    !Tr_meulage_bavure : Meulage de la bavure
    LOCAL CONST Robtarget Tr_meulage_bavure_0 := [[-118.3383671875,-114.213265625,120.94103125],[0.686050855165754,-0.669480714392343,0.19893041187492,-0.203854086086913],[0,0,0,0],[8.999999E+09,8.999999E+09,8.999999E+09,8.999999E+09,8.999999E+09,8.999999E+09]];
    LOCAL CONST Robtarget Tr_meulage_bavure_1 := [[-119.6316875,-113.9973125,120.9542265625],[0.684325266912173,-0.667622761472622,0.204761653370109,-0.209884355630412],[0,0,0,0],[8.999999E+09,8.999999E+09,8.999999E+09,8.999999E+09,8.999999E+09,8.999999E+09]];
    LOCAL CONST Robtarget Tr_meulage_bavure_2 := [[-123.489203125,-113.0502109375,120.9455703125],[0.678831233917672,-0.66176958949123,0.222117553220813,-0.227844154705838],[0,0,0,0],[8.999999E+09,8.999999E+09,8.999999E+09,8.999999E+09,8.999999E+09,8.999999E+09]];
    LOCAL CONST Robtarget Tr_meulage_bavure_3 := [[-123.584859375,-113.0222734375,120.9446484375],[0.668624934223721,-0.651045700458164,0.250641046300353,-0.257408739476203],[0,0,0,0],[8.999999E+09,8.999999E+09,8.999999E+09,8.999999E+09,8.999999E+09,8.999999E+09]];
    LOCAL CONST Robtarget Tr_meulage_bavure_4 := [[-125.8031953125,-111.60703125,120.8016875],[0.652172819034723,-0.634001173456056,0.28968410592264,-0.297986987877738],[0,0,0,0],[8.999999E+09,8.999999E+09,8.999999E+09,8.999999E+09,8.999999E+09,8.999999E+09]];
    LOCAL CONST Robtarget Tr_meulage_bavure_5 := [[-126.4752265625,-111.0076484375,120.7313359375],[0.627744539207993,-0.609028304977179,0.337572017036929,-0.347946045450712],[0,0,0,0],[8.999999E+09,8.999999E+09,8.999999E+09,8.999999E+09,8.999999E+09,8.999999E+09]];
    LOCAL CONST Robtarget Tr_meulage_bavure_6 := [[-126.8417890625,-109.187203125,120.45625],[0.594928081420455,-0.575888879676794,0.389993371636008,-0.402886766079456],[0,0,0,0],[8.999999E+09,8.999999E+09,8.999999E+09,8.999999E+09,8.999999E+09,8.999999E+09]];
    LOCAL CONST Robtarget Tr_meulage_bavure_7 := [[-127.4551015625,-107.313234375,120.181734375],[0.55678322484501,-0.537637245657738,0.439837894187461,-0.455501108066151],[0,0,0,0],[8.999999E+09,8.999999E+09,8.999999E+09,8.999999E+09,8.999999E+09,8.999999E+09]];
    LOCAL CONST Robtarget Tr_meulage_bavure_8 := [[-126.9923671875,-103.8465,119.6153203125],[0.519549603690322,-0.500370572095961,0.48044926250951,-0.498864717172559],[0,0,0,0],[8.999999E+09,8.999999E+09,8.999999E+09,8.999999E+09,8.999999E+09,8.999999E+09]];
    LOCAL CONST Robtarget Tr_meulage_bavure_9 := [[-126.982359375,-103.7414453125,119.5983046875],[0.489009720279578,-0.469707644324052,0.509165648687706,-0.530089204315714],[0,0,0,0],[8.999999E+09,8.999999E+09,8.999999E+09,8.999999E+09,8.999999E+09,8.999999E+09]];
    LOCAL CONST Robtarget Tr_meulage_bavure_10 := [[-126.968546875,-103.6983828125,119.5909765625],[0.467640365028404,-0.44800873567007,0.527122282578491,-0.550220647530287],[0,0,0,0],[8.999999E+09,8.999999E+09,8.999999E+09,8.999999E+09,8.999999E+09,8.999999E+09]];
    LOCAL CONST Robtarget Tr_meulage_bavure_11 := [[-126.9365390625,-103.55375,119.566875],[0.454927941273034,-0.434723512970439,0.536951278731924,-0.561906896013807],[0,0,0,0],[8.999999E+09,8.999999E+09,8.999999E+09,8.999999E+09,8.999999E+09,8.999999E+09]];
    LOCAL CONST Robtarget Tr_meulage_bavure_12 := [[-125.41084375,-97.252625,118.5122578125],[0.448816582731819,-0.427864419149345,0.541337479198651,-0.567846323846318],[0,0,0,0],[8.999999E+09,8.999999E+09,8.999999E+09,8.999999E+09,8.999999E+09,8.999999E+09]];
    LOCAL CONST Robtarget Tr_meulage_bavure_13 := [[-124.5225390625,-93.8810859375,117.945328125],[0.446998595891194,-0.425203405993345,0.54242876260288,-0.570232721179755],[0,0,0,0],[8.999999E+09,8.999999E+09,8.999999E+09,8.999999E+09,8.999999E+09,8.999999E+09]];
    LOCAL CONST Robtarget Tr_meulage_bavure_14 := [[-123.5930703125,-90.2569375,117.3368515625],[0.447502976011157,-0.424854620024497,0.541806054841724,-0.570688914595198],[0,0,0,0],[8.999999E+09,8.999999E+09,8.999999E+09,8.999999E+09,8.999999E+09,8.999999E+09]];
    LOCAL CONST Robtarget Tr_meulage_bavure_15 := [[-122.23978125,-84.399203125,116.3588359375],[0.448989970749093,-0.425524113227847,0.540477114320348,-0.57028214431484],[0,0,0,0],[8.999999E+09,8.999999E+09,8.999999E+09,8.999999E+09,8.999999E+09,8.999999E+09]];
    LOCAL CONST Robtarget Tr_meulage_bavure_16 := [[-121.5735078125,-81.584796875,115.88834375],[0.450680481375244,-0.426476052278341,0.539022241105553,-0.569614171289661],[0,0,0,0],[8.999999E+09,8.999999E+09,8.999999E+09,8.999999E+09,8.999999E+09,8.999999E+09]];
    LOCAL CONST Robtarget Tr_meulage_bavure_17 := [[-120.9896015625,-79.18940625,115.4872890625],[0.452134574382777,-0.427316386761855,0.537776039621201,-0.569009633891935],[0,0,0,0],[8.999999E+09,8.999999E+09,8.999999E+09,8.999999E+09,8.999999E+09,8.999999E+09]];
    LOCAL CONST Robtarget Tr_meulage_bavure_18 := [[-120.019578125,-75.11315625,114.805671875],[0.453213788071953,-0.427880207944664,0.536833179665065,-0.568617557908124],[0,0,0,0],[8.999999E+09,8.999999E+09,8.999999E+09,8.999999E+09,8.999999E+09,8.999999E+09]];
    LOCAL CONST Robtarget Tr_meulage_bavure_19 := [[-117.8866484375,-66.2634140625,113.3248515625],[0.453844832375933,-0.428071672477321,0.536242057569294,-0.568527894691176],[0,0,0,0],[8.999999E+09,8.999999E+09,8.999999E+09,8.999999E+09,8.999999E+09,8.999999E+09]];
    LOCAL CONST Robtarget Tr_meulage_bavure_20 := [[-117.3607109375,-63.81588671875,112.91765625],[0.453984641461937,-0.427853174272189,0.536036096461687,-0.568774920220648],[0,0,0,0],[8.999999E+09,8.999999E+09,8.999999E+09,8.999999E+09,8.999999E+09,8.999999E+09]];
    LOCAL CONST Robtarget Tr_meulage_bavure_21 := [[-116.8446015625,-61.71109375,112.565140625],[0.453678596601359,-0.42724510875903,0.536173528737094,-0.569346375336595],[0,0,0,0],[8.999999E+09,8.999999E+09,8.999999E+09,8.999999E+09,8.999999E+09,8.999999E+09]];
    LOCAL CONST Robtarget Tr_meulage_bavure_22 := [[-115.140578125,-54.66884375,111.3865234375],[0.453041728465808,-0.426338137315311,0.536560694775943,-0.570168050455988],[0,0,0,0],[8.999999E+09,8.999999E+09,8.999999E+09,8.999999E+09,8.999999E+09,8.999999E+09]];
    LOCAL CONST Robtarget Tr_meulage_bavure_23 := [[-114.799265625,-53.2905,111.1555546875],[0.452268427426111,-0.425270638734429,0.53703690263279,-0.571130036501761],[0,0,0,0],[8.999999E+09,8.999999E+09,8.999999E+09,8.999999E+09,8.999999E+09,8.999999E+09]];
    LOCAL CONST Robtarget Tr_meulage_bavure_24 := [[-113.7839921875,-49.33275390625,110.4910625],[0.451566366033952,-0.424226454223766,0.537443001430753,-0.572079323885006],[0,0,0,0],[8.999999E+09,8.999999E+09,8.999999E+09,8.999999E+09,8.999999E+09,8.999999E+09]];
    LOCAL CONST Robtarget Tr_meulage_bavure_25 := [[-113.1937265625,-47.288171875,110.1453671875],[0.451120847088053,-0.423372780939976,0.537640181481525,-0.572877390842247],[0,0,0,0],[8.999999E+09,8.999999E+09,8.999999E+09,8.999999E+09,8.999999E+09,8.999999E+09]];
    LOCAL CONST Robtarget Tr_meulage_bavure_26 := [[-113.1840546875,-47.07825,110.1117421875],[0.451087827748652,-0.422822590793089,0.537504839546807,-0.573436461899472],[0,0,0,0],[8.999999E+09,8.999999E+09,8.999999E+09,8.999999E+09,8.999999E+09,8.999999E+09]];
    LOCAL CONST Robtarget Tr_meulage_bavure_27 := [[-113.1511875,-46.92472265625,110.086203125],[0.451550947267371,-0.42264652281122,0.536974925089128,-0.573698168554729],[0,0,0,0],[8.999999E+09,8.999999E+09,8.999999E+09,8.999999E+09,8.999999E+09,8.999999E+09]];
    LOCAL CONST Robtarget Tr_meulage_bavure_28 := [[-113.0726328125,-46.59278515625,110.03071875],[0.452529309704206,-0.422852528909516,0.536034635844252,-0.573654801974831],[0,0,0,0],[8.999999E+09,8.999999E+09,8.999999E+09,8.999999E+09,8.999999E+09,8.999999E+09]];
    LOCAL CONST Robtarget Tr_meulage_bavure_29 := [[-112.882953125,-45.70284765625,109.8827109375],[0.454003221451682,-0.423425757175937,0.534699883466271,-0.573312949175784],[0,0,0,0],[8.999999E+09,8.999999E+09,8.999999E+09,8.999999E+09,8.999999E+09,8.999999E+09]];
    LOCAL CONST Robtarget Tr_meulage_bavure_30 := [[-111.1116875,-38.37715625,108.6567109375],[0.45587227688014,-0.42428239303802,0.533047220326503,-0.572735173559505],[0,0,0,0],[8.999999E+09,8.999999E+09,8.999999E+09,8.999999E+09,8.999999E+09,8.999999E+09]];
    LOCAL CONST Robtarget Tr_meulage_bavure_31 := [[-110.378484375,-35.3485,108.1498125],[0.457963860044262,-0.425242350058571,0.531197869017026,-0.572072434715914],[0,0,0,0],[8.999999E+09,8.999999E+09,8.999999E+09,8.999999E+09,8.999999E+09,8.999999E+09]];
    LOCAL CONST Robtarget Tr_meulage_bavure_32 := [[-110.08765625,-34.151265625,107.9493984375],[0.460081625202868,-0.42617821048254,0.529314222994711,-0.57142233452683],[0,0,0,0],[8.999999E+09,8.999999E+09,8.999999E+09,8.999999E+09,8.999999E+09,8.999999E+09]];
    LOCAL CONST Robtarget Tr_meulage_bavure_33 := [[-109.7187734375,-32.0638203125,107.60503125],[0.462073195478615,-0.426964804841995,0.527515145883789,-0.570891573163962],[0,0,0,0],[8.999999E+09,8.999999E+09,8.999999E+09,8.999999E+09,8.999999E+09,8.999999E+09]];
    LOCAL CONST Robtarget Tr_meulage_bavure_34 := [[-108.910796875,-29.1835546875,107.11890625],[0.464014309413054,-0.427683254437214,0.525747907017036,-0.570409408058042],[0,0,0,0],[8.999999E+09,8.999999E+09,8.999999E+09,8.999999E+09,8.999999E+09,8.999999E+09]];
    LOCAL CONST Robtarget Tr_meulage_bavure_35 := [[-108.8531484375,-28.931478515625,107.0768359375],[0.466195342276825,-0.42865743936496,0.523810839636805,-0.569681408153237],[0,0,0,0],[8.999999E+09,8.999999E+09,8.999999E+09,8.999999E+09,8.999999E+09,8.999999E+09]];
    LOCAL CONST Robtarget Tr_meulage_bavure_36 := [[-107.29965625,-21.97473828125,105.917296875],[0.468990155250694,-0.430255580003777,0.521426305856013,-0.568368698746593],[0,0,0,0],[8.999999E+09,8.999999E+09,8.999999E+09,8.999999E+09,8.999999E+09,8.999999E+09]];
    LOCAL CONST Robtarget Tr_meulage_bavure_37 := [[-107.0385390625,-20.856716796875,105.7305234375],[0.472580332865585,-0.43267861722955,0.518456365236538,-0.566268523340911],[0,0,0,0],[8.999999E+09,8.999999E+09,8.999999E+09,8.999999E+09,8.999999E+09,8.999999E+09]];
    LOCAL CONST Robtarget Tr_meulage_bavure_38 := [[-104.5382890625,-10.910146484375,104.06240625],[0.476562728941706,-0.435590355351763,0.51520207784131,-0.563662866167495],[0,0,0,0],[8.999999E+09,8.999999E+09,8.999999E+09,8.999999E+09,8.999999E+09,8.999999E+09]];
    LOCAL CONST Robtarget Tr_meulage_bavure_39 := [[-104.4991640625,-10.7461748046875,104.034984375],[0.479902988264319,-0.438094538801173,0.512468875028467,-0.561375052041522],[0,0,0,0],[8.999999E+09,8.999999E+09,8.999999E+09,8.999999E+09,8.999999E+09,8.999999E+09]];
    LOCAL CONST Robtarget Tr_meulage_bavure_40 := [[-102.5526875,-2.02845654296875,102.5819296875],[0.481332254936157,-0.439057645671762,0.511266939372169,-0.560494211245986],[0,0,0,0],[8.999999E+09,8.999999E+09,8.999999E+09,8.999999E+09,8.999999E+09,8.999999E+09]];
    LOCAL CONST Robtarget Tr_meulage_bavure_41 := [[-101.6165234375,1.70711413574219,101.955546875],[0.480183207612183,-0.43789436821085,0.512136374957438,-0.561594998964512],[0,0,0,0],[8.999999E+09,8.999999E+09,8.999999E+09,8.999999E+09,8.999999E+09,8.999999E+09]];
    LOCAL CONST Robtarget Tr_meulage_bavure_42 := [[-101.1611328125,3.43966796875,101.6642578125],[0.476920224473277,-0.435042441138407,0.514698164897639,-0.564243717685628],[0,0,0,0],[8.999999E+09,8.999999E+09,8.999999E+09,8.999999E+09,8.999999E+09,8.999999E+09]];
    LOCAL CONST Robtarget Tr_meulage_bavure_43 := [[-100.8461484375,4.85256787109375,101.4287734375],[0.472734357170233,-0.431608523188393,0.518007726848779,-0.567366112124211],[0,0,0,0],[8.999999E+09,8.999999E+09,8.999999E+09,8.999999E+09,8.999999E+09,8.999999E+09]];
    LOCAL CONST Robtarget Tr_meulage_bavure_44 := [[-100.4778515625,6.11641552734375,101.2149609375],[0.468758061313262,-0.428596753674646,0.521190056104333,-0.570027743282158],[0,0,0,0],[8.999999E+09,8.999999E+09,8.999999E+09,8.999999E+09,8.999999E+09,8.999999E+09]];
    LOCAL CONST Robtarget Tr_meulage_bavure_45 := [[-98.949234375,12.3987919921875,100.1632109375],[0.465580433550666,-0.426541653391156,0.52381904607302,-0.57176103818664],[0,0,0,0],[8.999999E+09,8.999999E+09,8.999999E+09,8.999999E+09,8.999999E+09,8.999999E+09]];
    LOCAL CONST Robtarget Tr_meulage_bavure_46 := [[-98.946515625,12.4088896484375,100.1615078125],[0.463203648755925,-0.425433029969794,0.52590814768651,-0.572599106694083],[0,0,0,0],[8.999999E+09,8.999999E+09,8.999999E+09,8.999999E+09,8.999999E+09,8.999999E+09]];
    LOCAL CONST Robtarget Tr_meulage_bavure_47 := [[-98.9428984375,12.4211572265625,100.1594296875],[0.46136081678198,-0.425012224249353,0.52766013929917,-0.572787555182253],[0,0,0,0],[8.999999E+09,8.999999E+09,8.999999E+09,8.999999E+09,8.999999E+09,8.999999E+09]];
    LOCAL CONST Robtarget Tr_meulage_bavure_48 := [[-98.9408671875,12.4388505859375,100.1565546875],[0.459746710263078,-0.424953330010414,0.529289634765119,-0.572625630098361],[0,0,0,0],[8.999999E+09,8.999999E+09,8.999999E+09,8.999999E+09,8.999999E+09,8.999999E+09]];
    LOCAL CONST Robtarget Tr_meulage_bavure_49 := [[-98.0083671875,16.6191640625,99.4598203125],[0.458190074419762,-0.425093454423347,0.530921938474095,-0.572258076357642],[0,0,0,0],[8.999999E+09,8.999999E+09,8.999999E+09,8.999999E+09,8.999999E+09,8.999999E+09]];
    LOCAL CONST Robtarget Tr_meulage_bavure_50 := [[-96.079359375,24.08840625,98.2052734375],[0.456753787612165,-0.425469707942997,0.532503116209528,-0.571657184291411],[0,0,0,0],[8.999999E+09,8.999999E+09,8.999999E+09,8.999999E+09,8.999999E+09,8.999999E+09]];
    LOCAL CONST Robtarget Tr_meulage_bavure_51 := [[-95.8122734375,25.151359375,98.027015625],[0.455596372896057,-0.426153186542171,0.533890319641322,-0.570777130933955],[0,0,0,0],[8.999999E+09,8.999999E+09,8.999999E+09,8.999999E+09,8.999999E+09,8.999999E+09]];
    LOCAL CONST Robtarget Tr_meulage_bavure_52 := [[-95.2577265625,27.313193359375,97.664046875],[0.45490178675266,-0.427311721276675,0.534940713644946,-0.569480017343751],[0,0,0,0],[8.999999E+09,8.999999E+09,8.999999E+09,8.999999E+09,8.999999E+09,8.999999E+09]];
    LOCAL CONST Robtarget Tr_meulage_bavure_53 := [[-94.4360390625,30.77109765625,97.085875],[0.454779594808474,-0.429012269576818,0.535553743534282,-0.56772016036495],[0,0,0,0],[8.999999E+09,8.999999E+09,8.999999E+09,8.999999E+09,8.999999E+09,8.999999E+09]];
    LOCAL CONST Robtarget Tr_meulage_bavure_54 := [[-94.0114609375,32.252177734375,96.8355703125],[0.455207955563008,-0.431195769741176,0.53572439451611,-0.565557511195643],[0,0,0,0],[8.999999E+09,8.999999E+09,8.999999E+09,8.999999E+09,8.999999E+09,8.999999E+09]];
    LOCAL CONST Robtarget Tr_meulage_bavure_55 := [[-93.2463671875,35.4615625,96.2988515625],[0.456074988327069,-0.43371784999866,0.535516993928133,-0.563121639460943],[0,0,0,0],[8.999999E+09,8.999999E+09,8.999999E+09,8.999999E+09,8.999999E+09,8.999999E+09]];
    LOCAL CONST Robtarget Tr_meulage_bavure_56 := [[-93.194546875,35.67014453125,96.2638984375],[0.457208597541458,-0.43636505275056,0.535044086377509,-0.560601163666854],[0,0,0,0],[8.999999E+09,8.999999E+09,8.999999E+09,8.999999E+09,8.999999E+09,8.999999E+09]];
    LOCAL CONST Robtarget Tr_meulage_bavure_57 := [[-93.1386484375,35.9594765625,96.2159921875],[0.458409657654475,-0.438922204807347,0.534453391732331,-0.558182278437762],[0,0,0,0],[8.999999E+09,8.999999E+09,8.999999E+09,8.999999E+09,8.999999E+09,8.999999E+09]];
    LOCAL CONST Robtarget Tr_meulage_bavure_58 := [[-92.5275390625,38.9375234375,95.7215859375],[0.459506167395724,-0.441171445416588,0.533872270361757,-0.556059562289072],[0,0,0,0],[8.999999E+09,8.999999E+09,8.999999E+09,8.999999E+09,8.999999E+09,8.999999E+09]];
    LOCAL CONST Robtarget Tr_meulage_bavure_59 := [[-92.266359375,40.06748046875,95.532921875],[0.460368536558143,-0.442902630890194,0.533393105421244,-0.554427511210384],[0,0,0,0],[8.999999E+09,8.999999E+09,8.999999E+09,8.999999E+09,8.999999E+09,8.999999E+09]];
    LOCAL CONST Robtarget Tr_meulage_bavure_60 := [[-90.608828125,46.17075390625,94.504828125],[0.460872183039202,-0.443983920750736,0.533123575247056,-0.553402532096918],[0,0,0,0],[8.999999E+09,8.999999E+09,8.999999E+09,8.999999E+09,8.999999E+09,8.999999E+09]];
    LOCAL CONST Robtarget Tr_meulage_bavure_61 := [[-90.312,48.11851953125,94.1852421875],[0.460979140838118,-0.444317386401172,0.533088683402381,-0.553079331996865],[0,0,0,0],[8.999999E+09,8.999999E+09,8.999999E+09,8.999999E+09,8.999999E+09,8.999999E+09]];
    LOCAL CONST Robtarget Tr_meulage_bavure_62 := [[-89.532015625,51.1954296875,93.668984375],[0.460726685185921,-0.443885486945191,0.533249554937321,-0.55348126273269],[0,0,0,0],[8.999999E+09,8.999999E+09,8.999999E+09,8.999999E+09,8.999999E+09,8.999999E+09]];
    LOCAL CONST Robtarget Tr_meulage_bavure_63 := [[-89.2893828125,52.2261328125,93.4967265625],[0.460233582250482,-0.442738162232384,0.533493028375766,-0.55457475433564],[0,0,0,0],[8.999999E+09,8.999999E+09,8.999999E+09,8.999999E+09,8.999999E+09,8.999999E+09]];
    LOCAL CONST Robtarget Tr_meulage_bavure_64 := [[-88.731390625,54.5765625,93.1037421875],[0.459639772094917,-0.440983470946271,0.533692406557432,-0.556270863378309],[0,0,0,0],[8.999999E+09,8.999999E+09,8.999999E+09,8.999999E+09,8.999999E+09,8.999999E+09]];
    LOCAL CONST Robtarget Tr_meulage_bavure_65 := [[-88.2320078125,56.53207421875,92.7755],[0.459072396008484,-0.438747093231614,0.533735951958913,-0.558461688023764],[0,0,0,0],[8.999999E+09,8.999999E+09,8.999999E+09,8.999999E+09,8.999999E+09,8.999999E+09]];
    LOCAL CONST Robtarget Tr_meulage_bavure_66 := [[-87.8954453125,57.63062890625,92.589046875],[0.458668017025218,-0.436081274379201,0.533484341816746,-0.561116056917213],[0,0,0,0],[8.999999E+09,8.999999E+09,8.999999E+09,8.999999E+09,8.999999E+09,8.999999E+09]];
    LOCAL CONST Robtarget Tr_meulage_bavure_67 := [[-87.7511875,58.13453515625,92.5038984375],[0.458509352199886,-0.433039573706918,0.532852713223189,-0.564193129663644],[0,0,0,0],[8.999999E+09,8.999999E+09,8.999999E+09,8.999999E+09,8.999999E+09,8.999999E+09]];
    LOCAL CONST Robtarget Tr_meulage_bavure_68 := [[-87.3662265625,59.9265,92.2057734375],[0.458659369679696,-0.429695408082701,0.531782315047372,-0.567627526006732],[0,0,0,0],[8.999999E+09,8.999999E+09,8.999999E+09,8.999999E+09,8.999999E+09,8.999999E+09]];
    LOCAL CONST Robtarget Tr_meulage_bavure_69 := [[-86.5865,63.57164453125,91.599453125],[0.459204100392526,-0.426106225696507,0.530188688699514,-0.571371186690805],[0,0,0,0],[8.999999E+09,8.999999E+09,8.999999E+09,8.999999E+09,8.999999E+09,8.999999E+09]];
    LOCAL CONST Robtarget Tr_meulage_bavure_70 := [[-86.236421875,64.864671875,91.3816875],[0.460224347850539,-0.422350837320893,0.528002030606232,-0.575349611571593],[0,0,0,0],[8.999999E+09,8.999999E+09,8.999999E+09,8.999999E+09,8.999999E+09,8.999999E+09]];
    LOCAL CONST Robtarget Tr_meulage_bavure_71 := [[-85.6366953125,67.1714609375,90.99409375],[0.461768432066829,-0.418464834045386,0.525176508528011,-0.579522849164929],[0,0,0,0],[8.999999E+09,8.999999E+09,8.999999E+09,8.999999E+09,8.999999E+09,8.999999E+09]];
    LOCAL CONST Robtarget Tr_meulage_bavure_72 := [[-84.1965390625,72.4226796875,90.109015625],[0.463744433304246,-0.414405956077751,0.521785359699143,-0.583908248400589],[0,0,0,0],[8.999999E+09,8.999999E+09,8.999999E+09,8.999999E+09,8.999999E+09,8.999999E+09]];
    LOCAL CONST Robtarget Tr_meulage_bavure_73 := [[-83.8633984375,73.8428125,89.87171875],[0.465931695568103,-0.410032056336984,0.517993747117799,-0.588611795488298],[0,0,0,0],[8.999999E+09,8.999999E+09,8.999999E+09,8.999999E+09,8.999999E+09,8.999999E+09]];
    LOCAL CONST Robtarget Tr_meulage_bavure_74 := [[-83.605078125,75.00646875,89.6778203125],[0.467962555054418,-0.405048292550795,0.514045111921415,-0.593889342115453],[0,0,0,0],[8.999999E+09,8.999999E+09,8.999999E+09,8.999999E+09,8.999999E+09,8.999999E+09]];
    LOCAL CONST Robtarget Tr_meulage_bavure_75 := [[-81.8162890625,82.1775546875,88.475671875],[0.469194146092542,-0.399043561537106,0.510383916210831,-0.600107779770907],[0,0,0,0],[8.999999E+09,8.999999E+09,8.999999E+09,8.999999E+09,8.999999E+09,8.999999E+09]];
    LOCAL CONST Robtarget Tr_meulage_bavure_76 := [[-81.625515625,82.8586640625,88.3607265625],[0.468788571727036,-0.391479701480755,0.507540713671349,-0.60776915215618],[0,0,0,0],[8.999999E+09,8.999999E+09,8.999999E+09,8.999999E+09,8.999999E+09,8.999999E+09]];
    LOCAL CONST Robtarget Tr_meulage_bavure_77 := [[-81.2855859375,84.3813671875,88.1069296875],[0.465684225577351,-0.381640921964858,0.506092770843089,-0.617542319222416],[0,0,0,0],[8.999999E+09,8.999999E+09,8.999999E+09,8.999999E+09,8.999999E+09,8.999999E+09]];
    LOCAL CONST Robtarget Tr_meulage_bavure_78 := [[-80.4661328125,88.0701328125,87.4922421875],[0.458504368662927,-0.36869083310866,0.506711104697416,-0.630146546348527],[0,0,0,0],[8.999999E+09,8.999999E+09,8.999999E+09,8.999999E+09,8.999999E+09,8.999999E+09]];
    LOCAL CONST Robtarget Tr_meulage_bavure_79 := [[-79.9652890625,90.3361328125,87.1147421875],[0.44558542121353,-0.351622898811277,0.510011593834459,-0.646299577276629],[0,0,0,0],[8.999999E+09,8.999999E+09,8.999999E+09,8.999999E+09,8.999999E+09,8.999999E+09]];
    LOCAL CONST Robtarget Tr_meulage_bavure_80 := [[-79.203953125,93.197921875,86.6332578125],[0.424956455516055,-0.329268592448,0.516452117066445,-0.666536882490483],[0,0,0,0],[8.999999E+09,8.999999E+09,8.999999E+09,8.999999E+09,8.999999E+09,8.999999E+09]];
    LOCAL CONST Robtarget Tr_meulage_bavure_81 := [[-78.5163515625,94.6883203125,86.371828125],[0.394497826109862,-0.30038935975108,0.526094666045292,-0.690913959984615],[0,0,0,0],[8.999999E+09,8.999999E+09,8.999999E+09,8.999999E+09,8.999999E+09,8.999999E+09]];
    LOCAL CONST Robtarget Tr_meulage_bavure_82 := [[-78.391578125,95.044234375,86.31084375],[0.352599084750227,-0.264168107079915,0.538261179634226,-0.718445543610571],[0,0,0,0],[8.999999E+09,8.999999E+09,8.999999E+09,8.999999E+09,8.999999E+09,8.999999E+09]];
    LOCAL CONST Robtarget Tr_meulage_bavure_83 := [[-76.9551328125,96.9148125,85.961703125],[0.299658971487937,-0.221242446743258,0.551223833743886,-0.746597994692284],[0,0,0,0],[8.999999E+09,8.999999E+09,8.999999E+09,8.999999E+09,8.999999E+09,8.999999E+09]];
    LOCAL CONST Robtarget Tr_meulage_bavure_84 := [[-76.393328125,97.6691953125,85.8215390625],[0.239664457549089,-0.174696559641749,0.56254110325317,-0.771744495923193],[0,0,0,0],[8.999999E+09,8.999999E+09,8.999999E+09,8.999999E+09,8.999999E+09,8.999999E+09]];
    LOCAL CONST Robtarget Tr_meulage_bavure_85 := [[-76.30184375,97.74853125,85.805609375],[0.179677116560747,-0.129574269659455,0.570386700540112,-0.790939728597318],[0,0,0,0],[8.999999E+09,8.999999E+09,8.999999E+09,8.999999E+09,8.999999E+09,8.999999E+09]];
    LOCAL CONST Robtarget Tr_meulage_bavure_86 := [[-76.1692890625,97.7941953125,85.793515625],[0.126758018316264,-0.0906463340687071,0.57457749340916,-0.803477660535802],[0,0,0,0],[8.999999E+09,8.999999E+09,8.999999E+09,8.999999E+09,8.999999E+09,8.999999E+09]];
    LOCAL CONST Robtarget Tr_meulage_bavure_87 := [[-70.1861015625,99.2918203125,85.3367578125],[0.0851219950592498,-0.0605101151073412,0.576221284093186,-0.810593488553189],[0,0,0,0],[8.999999E+09,8.999999E+09,8.999999E+09,8.999999E+09,8.999999E+09,8.999999E+09]];
    LOCAL CONST Robtarget Tr_meulage_bavure_88 := [[-69.7351015625,99.25803125,85.325578125],[0.0562665210316202,-0.039860160076473,0.576686891338161,-0.814050044904123],[0,0,0,0],[8.999999E+09,8.999999E+09,8.999999E+09,8.999999E+09,8.999999E+09,8.999999E+09]];
    LOCAL CONST Robtarget Tr_meulage_bavure_89 := [[-66.7805,98.331390625,85.3641015625],[0.0407211958690712,-0.0288206439174172,0.576983784482189,-0.815230560722418],[0,0,0,0],[8.999999E+09,8.999999E+09,8.999999E+09,8.999999E+09,8.999999E+09,8.999999E+09]];
    LOCAL CONST Robtarget Tr_meulage_bavure_90 := [[-66.1347265625,98.1061640625,85.3761171875],[0.0389424577542935,-0.0276044605202579,0.57764016404893,-0.81489466780742],[0,0,0,0],[8.999999E+09,8.999999E+09,8.999999E+09,8.999999E+09,8.999999E+09,8.999999E+09]];
    LOCAL CONST Robtarget Tr_meulage_bavure_91 := [[-66.04090625,98.0874140625,85.3756484375],[0.0513935581339885,-0.0365740111652439,0.578658418714526,-0.813126975533598],[0,0,0,0],[8.999999E+09,8.999999E+09,8.999999E+09,8.999999E+09,8.999999E+09,8.999999E+09]];
    LOCAL CONST Robtarget Tr_meulage_bavure_92 := [[-65.928109375,98.0747265625,85.3735234375],[0.0777355817984993,-0.0556591700658173,0.579497359879816,-0.809346678502084],[0,0,0,0],[8.999999E+09,8.999999E+09,8.999999E+09,8.999999E+09,8.999999E+09,8.999999E+09]];
    LOCAL CONST Robtarget Tr_meulage_bavure_93 := [[-59.409203125,97.3848984375,85.2438203125],[0.115751958971051,-0.0835530618569988,0.579286121715875,-0.802525986517612],[0,0,0,0],[8.999999E+09,8.999999E+09,8.999999E+09,8.999999E+09,8.999999E+09,8.999999E+09]];
    LOCAL CONST Robtarget Tr_meulage_bavure_94 := [[-57.24732421875,98.220609375,85.03209375],[0.160944636884409,-0.117316903909768,0.577244865637887,-0.791910306164701],[0,0,0,0],[8.999999E+09,8.999999E+09,8.999999E+09,8.999999E+09,8.999999E+09,8.999999E+09]];
    LOCAL CONST Robtarget Tr_meulage_bavure_95 := [[-56.4332109375,98.4947265625,84.958796875],[0.207665394146208,-0.153077424336631,0.573265800188772,-0.777694482792883],[0,0,0,0],[8.999999E+09,8.999999E+09,8.999999E+09,8.999999E+09,8.999999E+09,8.999999E+09]];
    LOCAL CONST Robtarget Tr_meulage_bavure_96 := [[-55.53553125,99.220390625,84.8108671875],[0.251613536654352,-0.187761221557354,0.567825707991313,-0.76092727457737],[0,0,0,0],[8.999999E+09,8.999999E+09,8.999999E+09,8.999999E+09,8.999999E+09,8.999999E+09]];
    LOCAL CONST Robtarget Tr_meulage_bavure_97 := [[-53.341171875,100.7332109375,84.490640625],[0.291312103215093,-0.220224084273424,0.561395303595543,-0.742612903420887],[0,0,0,0],[8.999999E+09,8.999999E+09,8.999999E+09,8.999999E+09,8.999999E+09,8.999999E+09]];
    LOCAL CONST Robtarget Tr_meulage_bavure_98 := [[-52.63539453125,101.5195234375,84.3401328125],[0.327279332426981,-0.250733708213391,0.554063309911272,-0.723211376253082],[0,0,0,0],[8.999999E+09,8.999999E+09,8.999999E+09,8.999999E+09,8.999999E+09,8.999999E+09]];
    LOCAL CONST Robtarget Tr_meulage_bavure_99 := [[-51.506703125,103.359203125,84.007171875],[0.360348635928472,-0.27975839301075,0.545709241046459,-0.70291217542523],[0,0,0,0],[8.999999E+09,8.999999E+09,8.999999E+09,8.999999E+09,8.999999E+09,8.999999E+09]];
    LOCAL CONST Robtarget Tr_meulage_bavure_100 := [[-51.01259375,104.2113671875,83.8539921875],[0.390475580502164,-0.307089551771606,0.536508519320608,-0.682190176505512],[0,0,0,0],[8.999999E+09,8.999999E+09,8.999999E+09,8.999999E+09,8.999999E+09,8.999999E+09]];
    LOCAL CONST Robtarget Tr_meulage_bavure_101 := [[-50.18411328125,106.450515625,83.468734375],[0.416684903465605,-0.331735568044641,0.527153117018851,-0.662144089557],[0,0,0,0],[8.999999E+09,8.999999E+09,8.999999E+09,8.999999E+09,8.999999E+09,8.999999E+09]];
    LOCAL CONST Robtarget Tr_meulage_bavure_102 := [[-49.38801171875,109.3609296875,82.978265625],[0.437803548895459,-0.352489711076903,0.518692994906855,-0.644233368581619],[0,0,0,0],[8.999999E+09,8.999999E+09,8.999999E+09,8.999999E+09,8.999999E+09,8.999999E+09]];
    LOCAL CONST Robtarget Tr_meulage_bavure_103 := [[-48.01431640625,114.901421875,82.04978125],[0.453254188188437,-0.36860094977623,0.51206645146158,-0.629668110992805],[0,0,0,0],[8.999999E+09,8.999999E+09,8.999999E+09,8.999999E+09,8.999999E+09,8.999999E+09]];
    LOCAL CONST Robtarget Tr_meulage_bavure_104 := [[-46.40897265625,122.5723046875,80.7751484375],[0.463240725750373,-0.379966222084329,0.507760113438182,-0.619042298459866],[0,0,0,0],[8.999999E+09,8.999999E+09,8.999999E+09,8.999999E+09,8.999999E+09,8.999999E+09]];
    LOCAL CONST Robtarget Tr_meulage_bavure_105 := [[-45.1870078125,127.51,79.9477578125],[0.468322830887073,-0.386845595799563,0.505896567909685,-0.612448262025129],[0,0,0,0],[8.999999E+09,8.999999E+09,8.999999E+09,8.999999E+09,8.999999E+09,8.999999E+09]];
    LOCAL CONST Robtarget Tr_meulage_bavure_106 := [[-44.53079296875,130.387484375,79.467640625],[0.469099575531706,-0.389577660536901,0.506366449142727,-0.609727688258581],[0,0,0,0],[8.999999E+09,8.999999E+09,8.999999E+09,8.999999E+09,8.999999E+09,8.999999E+09]];
    LOCAL CONST Robtarget Tr_meulage_bavure_107 := [[-44.1889296875,131.99715625,79.1999921875],[0.465738311234576,-0.388207522142932,0.509162028735586,-0.610849223371752],[0,0,0,0],[8.999999E+09,8.999999E+09,8.999999E+09,8.999999E+09,8.999999E+09,8.999999E+09]];
    LOCAL CONST Robtarget Tr_meulage_bavure_108 := [[-43.83968359375,133.83725,78.895546875],[0.457668427312981,-0.382266322767619,0.5146054314194,-0.616111450203807],[0,0,0,0],[8.999999E+09,8.999999E+09,8.999999E+09,8.999999E+09,8.999999E+09,8.999999E+09]];
    LOCAL CONST Robtarget Tr_meulage_bavure_109 := [[-43.1372890625,137.40815625,78.303828125],[0.443597928270363,-0.370702333935445,0.523232407122641,-0.626121797884168],[0,0,0,0],[8.999999E+09,8.999999E+09,8.999999E+09,8.999999E+09,8.999999E+09,8.999999E+09]];
    LOCAL CONST Robtarget Tr_meulage_bavure_110 := [[-42.73471875,138.825703125,78.0643984375],[0.421721082233463,-0.352092749806372,0.535511575512922,-0.641412017992564],[0,0,0,0],[8.999999E+09,8.999999E+09,8.999999E+09,8.999999E+09,8.999999E+09,8.999999E+09]];
    LOCAL CONST Robtarget Tr_meulage_bavure_111 := [[-41.463578125,141.106890625,77.6562421875],[0.390202884755249,-0.325066577310493,0.551375820421673,-0.661859602709404],[0,0,0,0],[8.999999E+09,8.999999E+09,8.999999E+09,8.999999E+09,8.999999E+09,8.999999E+09]];
    LOCAL CONST Robtarget Tr_meulage_bavure_112 := [[-41.4130546875,141.188203125,77.6415078125],[0.347936130419601,-0.288923825160768,0.569781097610185,-0.686158125514256],[0,0,0,0],[8.999999E+09,8.999999E+09,8.999999E+09,8.999999E+09,8.999999E+09,8.999999E+09]];
    LOCAL CONST Robtarget Tr_meulage_bavure_113 := [[-39.915421875,142.683203125,77.3496484375],[0.295595742770883,-0.24448198254045,0.588580708467148,-0.711635065668585],[0,0,0,0],[8.999999E+09,8.999999E+09,8.999999E+09,8.999999E+09,8.999999E+09,8.999999E+09]];
    LOCAL CONST Robtarget Tr_meulage_bavure_114 := [[-39.54890234375,142.982109375,77.288828125],[0.236075941486186,-0.194365051857047,0.605161963355346,-0.735030186166474],[0,0,0,0],[8.999999E+09,8.999999E+09,8.999999E+09,8.999999E+09,8.999999E+09,8.999999E+09]];
    LOCAL CONST Robtarget Tr_meulage_bavure_115 := [[-38.14555859375,143.671671875,77.1280859375],[0.173782757830943,-0.142382823046795,0.617561581976808,-0.753753525529532],[0,0,0,0],[8.999999E+09,8.999999E+09,8.999999E+09,8.999999E+09,8.999999E+09,8.999999E+09]];
    LOCAL CONST Robtarget Tr_meulage_bavure_116 := [[-35.973265625,143.826484375,77.023890625],[0.113224092615185,-0.0923115627947642,0.625119681239126,-0.766736111288199],[0,0,0,0],[8.999999E+09,8.999999E+09,8.999999E+09,8.999999E+09,8.999999E+09,8.999999E+09]];
    LOCAL CONST Robtarget Tr_meulage_bavure_117 := [[-33.6576875,143.801609375,76.9429296875],[0.0581064457668376,-0.0471486693648434,0.628320307415449,-0.774347619113551],[0,0,0,0],[8.999999E+09,8.999999E+09,8.999999E+09,8.999999E+09,8.999999E+09,8.999999E+09]];
    LOCAL CONST Robtarget Tr_meulage_bavure_118 := [[-31.373509765625,143.500671875,76.9068671875],[0.0111183895401802,-0.0089817345611662,0.628336293346884,-0.777810524691846],[0,0,0,0],[8.999999E+09,8.999999E+09,8.999999E+09,8.999999E+09,8.999999E+09,8.999999E+09]];
    LOCAL CONST Robtarget Tr_meulage_bavure_119 := [[-29.340666015625,143.06459375,76.9014375],[0.0260475936494563,-0.0209598681049437,-0.626563297122989,0.778653094447371],[0,0,0,0],[8.999999E+09,8.999999E+09,8.999999E+09,8.999999E+09,8.999999E+09,8.999999E+09]];
    LOCAL CONST Robtarget Tr_meulage_bavure_120 := [[-28.516828125,142.861375,76.9034375],[0.052550119797892,-0.0421476810352239,-0.62424714525063,0.778317133011358],[0,0,0,0],[8.999999E+09,8.999999E+09,8.999999E+09,8.999999E+09,8.999999E+09,8.999999E+09]];
    LOCAL CONST Robtarget Tr_meulage_bavure_121 := [[-24.87820703125,141.7868125,76.940328125],[0.0681555721225083,-0.0545239673604753,-0.622307608491228,0.777891506179272],[0,0,0,0],[8.999999E+09,8.999999E+09,8.999999E+09,8.999999E+09,8.999999E+09,8.999999E+09]];
    LOCAL CONST Robtarget Tr_meulage_bavure_122 := [[-24.348373046875,141.62796875,76.9460703125],[0.0731750970994033,-0.0584338889801196,-0.621261356487815,0.777987925817664],[0,0,0,0],[8.999999E+09,8.999999E+09,8.999999E+09,8.999999E+09,8.999999E+09,8.999999E+09]];
    LOCAL CONST Robtarget Tr_meulage_bavure_123 := [[-16.3998828125,139.587953125,76.9779375],[0.0684288788643578,-0.0545900925375494,-0.621234731344755,0.77871998748274],[0,0,0,0],[8.999999E+09,8.999999E+09,8.999999E+09,8.999999E+09,8.999999E+09,8.999999E+09]];
    LOCAL CONST Robtarget Tr_meulage_bavure_124 := [[-13.923857421875,138.957875,76.9870078125],[0.05541922405158,-0.0442036046753149,-0.621992174469866,0.779807980106306],[0,0,0,0],[8.999999E+09,8.999999E+09,8.999999E+09,8.999999E+09,8.999999E+09,8.999999E+09]];
    LOCAL CONST Robtarget Tr_meulage_bavure_125 := [[-12.9184189453125,138.6723125,76.9953984375],[0.0365023876435811,-0.0291312957429179,-0.623092031215271,0.780753010843176],[0,0,0,0],[8.999999E+09,8.999999E+09,8.999999E+09,8.999999E+09,8.999999E+09,8.999999E+09]];
    LOCAL CONST Robtarget Tr_meulage_bavure_126 := [[-10.416712890625,138.40440625,76.946125],[0.0147352886266247,-0.0117744710468645,-0.624139069566195,0.781085561857151],[0,0,0,0],[8.999999E+09,8.999999E+09,8.999999E+09,8.999999E+09,8.999999E+09,8.999999E+09]];
    LOCAL CONST Robtarget Tr_meulage_bavure_127 := [[-7.6341181640625,138.29740625,76.8610546875],[0.00669345717475726,-0.00535866876042923,0.624949597056137,-0.780618013781093],[0,0,0,0],[8.999999E+09,8.999999E+09,8.999999E+09,8.999999E+09,8.999999E+09,8.999999E+09]];
    LOCAL CONST Robtarget Tr_meulage_bavure_128 := [[-7.003890625,138.375328125,76.82559375],[0.0252662795434682,-0.0202774222493153,0.625577820481968,-0.779488827236148],[0,0,0,0],[8.999999E+09,8.999999E+09,8.999999E+09,8.999999E+09,8.999999E+09,8.999999E+09]];
    LOCAL CONST Robtarget Tr_meulage_bavure_129 := [[-4.2065625,138.824890625,76.651765625],[0.0394890256379991,-0.0317840076765823,0.626205189755441,-0.778008646503063],[0,0,0,0],[8.999999E+09,8.999999E+09,8.999999E+09,8.999999E+09,8.999999E+09,8.999999E+09]];
    LOCAL CONST Robtarget Tr_meulage_bavure_130 := [[-3.08819189453125,139.11703125,76.5644609375],[0.0487026801204348,-0.0393285767742328,0.62702561509046,-0.776479355822439],[0,0,0,0],[8.999999E+09,8.999999E+09,8.999999E+09,8.999999E+09,8.999999E+09,8.999999E+09]];
    LOCAL CONST Robtarget Tr_meulage_bavure_131 := [[0.144217483520508,139.811859375,76.3358046875],[0.0526971924461445,-0.0427060956154171,0.62816192942171,-0.775120497555557],[0,0,0,0],[8.999999E+09,8.999999E+09,8.999999E+09,8.999999E+09,8.999999E+09,8.999999E+09]];
    LOCAL CONST Robtarget Tr_meulage_bavure_132 := [[1.4962587890625,140.145703125,76.2333203125],[0.0513418434197572,-0.0417639247550209,0.629651995329084,-0.774053069551062],[0,0,0,0],[8.999999E+09,8.999999E+09,8.999999E+09,8.999999E+09,8.999999E+09,8.999999E+09]];
    LOCAL CONST Robtarget Tr_meulage_bavure_133 := [[2.11551708984375,140.258703125,76.192703125],[0.0445551618241956,-0.0363835728929193,0.631454478537628,-0.77327635080425],[0,0,0,0],[8.999999E+09,8.999999E+09,8.999999E+09,8.999999E+09,8.999999E+09,8.999999E+09]];
    LOCAL CONST Robtarget Tr_meulage_bavure_134 := [[2.59485278320312,140.282734375,76.1713203125],[0.0325484123060889,-0.0266834182893128,0.633428591705382,-0.772655689977681],[0,0,0,0],[8.999999E+09,8.999999E+09,8.999999E+09,8.999999E+09,8.999999E+09,8.999999E+09]];
    LOCAL CONST Robtarget Tr_meulage_bavure_135 := [[4.8459609375,140.435734375,76.0645234375],[0.016128327313522,-0.0132743687836816,0.635346545438879,-0.771944580517504],[0,0,0,0],[8.999999E+09,8.999999E+09,8.999999E+09,8.999999E+09,8.999999E+09,8.999999E+09]];
    LOCAL CONST Robtarget Tr_meulage_bavure_136 := [[8.5892470703125,139.976234375,76.0000859375],[0.00313895726904941,-0.00259355609099817,-0.636949798648598,0.770894528723338],[0,0,0,0],[8.999999E+09,8.999999E+09,8.999999E+09,8.999999E+09,8.999999E+09,8.999999E+09]];
    LOCAL CONST Robtarget Tr_meulage_bavure_137 := [[8.9748994140625,139.931390625,75.9930546875],[0.0232174689920192,-0.0192565231275171,-0.638104546515992,0.769358644044677],[0,0,0,0],[8.999999E+09,8.999999E+09,8.999999E+09,8.999999E+09,8.999999E+09,8.999999E+09]];
    LOCAL CONST Robtarget Tr_meulage_bavure_138 := [[12.22753515625,139.095875,76.0062109375],[0.0420801009113633,-0.0350316256826077,-0.638845951825755,0.767383802373472],[0,0,0,0],[8.999999E+09,8.999999E+09,8.999999E+09,8.999999E+09,8.999999E+09,8.999999E+09]];
    LOCAL CONST Robtarget Tr_meulage_bavure_139 := [[20.129361328125,136.96746875,76.053796875],[0.0582116574303083,-0.0486380800342606,-0.639335111582264,0.76517733579079],[0,0,0,0],[8.999999E+09,8.999999E+09,8.999999E+09,8.999999E+09,8.999999E+09,8.999999E+09]];
    LOCAL CONST Robtarget Tr_meulage_bavure_140 := [[27.107314453125,135.27440625,76.0662578125],[0.0708465169456789,-0.0594060164556367,-0.639773486806526,0.762982032439138],[0,0,0,0],[8.999999E+09,8.999999E+09,8.999999E+09,8.999999E+09,8.999999E+09,8.999999E+09]];
    LOCAL CONST Robtarget Tr_meulage_bavure_141 := [[34.70656640625,133.395109375,76.0854609375],[0.079932014005928,-0.0672589989968302,-0.640320762912453,0.760970709537571],[0,0,0,0],[8.999999E+09,8.999999E+09,8.999999E+09,8.999999E+09,8.999999E+09,8.999999E+09]];
    LOCAL CONST Robtarget Tr_meulage_bavure_142 := [[37.201125,132.7344375,76.0986953125],[0.0859039191986607,-0.0725349289584913,-0.641058276494122,0.759212412231045],[0,0,0,0],[8.999999E+09,8.999999E+09,8.999999E+09,8.999999E+09,8.999999E+09,8.999999E+09]];
    LOCAL CONST Robtarget Tr_meulage_bavure_143 := [[46.7153203125,130.3923125,76.12103125],[0.0894422492300376,-0.0757858140360504,-0.642000991374565,0.757688142653454],[0,0,0,0],[8.999999E+09,8.999999E+09,8.999999E+09,8.999999E+09,8.999999E+09,8.999999E+09]];
    LOCAL CONST Robtarget Tr_meulage_bavure_144 := [[48.21742578125,130.0088125,76.126734375],[0.0912621789345908,-0.0776012626031111,-0.643121191260491,0.756336163415582],[0,0,0,0],[8.999999E+09,8.999999E+09,8.999999E+09,8.999999E+09,8.999999E+09,8.999999E+09]];
    LOCAL CONST Robtarget Tr_meulage_bavure_145 := [[49.14859375,129.777171875,76.1293046875],[0.0919775454937618,-0.0784953849823497,-0.644393710759899,0.755073076724699],[0,0,0,0],[8.999999E+09,8.999999E+09,8.999999E+09,8.999999E+09,8.999999E+09,8.999999E+09]];
    LOCAL CONST Robtarget Tr_meulage_bavure_146 := [[50.71092578125,129.4158671875,76.12928125],[0.0920557022147844,-0.078862484789295,-0.645792273562561,0.753829420750808],[0,0,0,0],[8.999999E+09,8.999999E+09,8.999999E+09,8.999999E+09,8.999999E+09,8.999999E+09]];
    LOCAL CONST Robtarget Tr_meulage_bavure_147 := [[60.2768984375,127.1642109375,76.135375],[0.0917503217506476,-0.0789185690849222,-0.647309358287523,0.75255852435916],[0,0,0,0],[8.999999E+09,8.999999E+09,8.999999E+09,8.999999E+09,8.999999E+09,8.999999E+09]];
    LOCAL CONST Robtarget Tr_meulage_bavure_148 := [[67.33846875,125.3770390625,76.1596953125],[0.0912404023297994,-0.0788186834643386,-0.648946618206938,0.75121973538867],[0,0,0,0],[8.999999E+09,8.999999E+09,8.999999E+09,8.999999E+09,8.999999E+09,8.999999E+09]];
    LOCAL CONST Robtarget Tr_meulage_bavure_149 := [[74.9421796875,123.49275,76.1795234375],[0.0907046142142524,-0.0787193343270008,-0.650702820965175,0.74977448486283],[0,0,0,0],[8.999999E+09,8.999999E+09,8.999999E+09,8.999999E+09,8.999999E+09,8.999999E+09]];
    LOCAL CONST Robtarget Tr_meulage_bavure_150 := [[87.3766796875,120.682203125,76.169015625],[0.0904347823724643,-0.0788779298263219,-0.65256216000458,0.748172740517667],[0,0,0,0],[8.999999E+09,8.999999E+09,8.999999E+09,8.999999E+09,8.999999E+09,8.999999E+09]];
    LOCAL CONST Robtarget Tr_meulage_bavure_151 := [[91.619484375,119.6658515625,76.1745234375],[0.0911610771075241,-0.0799394892455209,-0.654450780006731,0.746319980054361],[0,0,0,0],[8.999999E+09,8.999999E+09,8.999999E+09,8.999999E+09,8.999999E+09,8.999999E+09]];
    LOCAL CONST Robtarget Tr_meulage_bavure_152 := [[95.5963125,118.8018359375,76.1656328125],[0.0940991152991975,-0.0829913910208722,-0.65622770332569,0.744058456644516],[0,0,0,0],[8.999999E+09,8.999999E+09,8.999999E+09,8.999999E+09,8.999999E+09,8.999999E+09]];
    LOCAL CONST Robtarget Tr_meulage_bavure_153 := [[99.4676875,117.911234375,76.164828125],[0.101191232260942,-0.0897947741941448,-0.657629779392187,0.741093992889916],[0,0,0,0],[8.999999E+09,8.999999E+09,8.999999E+09,8.999999E+09,8.999999E+09,8.999999E+09]];
    LOCAL CONST Robtarget Tr_meulage_bavure_154 := [[107.5950546875,116.1329296875,76.14865625],[0.115244260446321,-0.102928800143851,-0.658131317520732,0.736876917424853],[0,0,0,0],[8.999999E+09,8.999999E+09,8.999999E+09,8.999999E+09,8.999999E+09,8.999999E+09]];
    LOCAL CONST Robtarget Tr_meulage_bavure_155 := [[112.979171875,115.017796875,76.12796875],[0.13984476900826,-0.12574767123199,-0.656702904430524,0.73032339348625],[0,0,0,0],[8.999999E+09,8.999999E+09,8.999999E+09,8.999999E+09,8.999999E+09,8.999999E+09]];
    LOCAL CONST Robtarget Tr_meulage_bavure_156 := [[113.9653515625,114.8439375,76.119359375],[0.178935786213355,-0.162025964488235,-0.65136379069437,0.719343300112073],[0,0,0,0],[8.999999E+09,8.999999E+09,8.999999E+09,8.999999E+09,8.999999E+09,8.999999E+09]];
    LOCAL CONST Robtarget Tr_meulage_bavure_157 := [[115.4251796875,114.414625,76.133875],[0.234959313352886,-0.214274470868327,-0.638857689704101,0.700529388754517],[0,0,0,0],[8.999999E+09,8.999999E+09,8.999999E+09,8.999999E+09,8.999999E+09,8.999999E+09]];
    LOCAL CONST Robtarget Tr_meulage_bavure_158 := [[117.4927265625,113.6852578125,76.1736640625],[0.304924715170675,-0.280074455246314,-0.615756183116296,0.670390588053423],[0,0,0,0],[8.999999E+09,8.999999E+09,8.999999E+09,8.999999E+09,8.999999E+09,8.999999E+09]];
    LOCAL CONST Robtarget Tr_meulage_bavure_159 := [[119.24453125,112.5415546875,76.2906875],[0.377537187575309,-0.349228030937531,-0.58236287838931,0.629570434724613],[0,0,0,0],[8.999999E+09,8.999999E+09,8.999999E+09,8.999999E+09,8.999999E+09,8.999999E+09]];
    LOCAL CONST Robtarget Tr_meulage_bavure_160 := [[120.623125,110.922359375,76.496765625],[0.439360227312934,-0.40921403360528,-0.545034820326455,0.585186730871209],[0,0,0,0],[8.999999E+09,8.999999E+09,8.999999E+09,8.999999E+09,8.999999E+09,8.999999E+09]];
    LOCAL CONST Robtarget Tr_meulage_bavure_161 := [[120.8545859375,110.5556328125,76.54640625],[0.484676318552652,-0.454385478603971,-0.511185750571127,0.545263084649164],[0,0,0,0],[8.999999E+09,8.999999E+09,8.999999E+09,8.999999E+09,8.999999E+09,8.999999E+09]];
    LOCAL CONST Robtarget Tr_meulage_bavure_162 := [[120.9014375,110.0289609375,76.62815625],[0.515595436675148,-0.486334352297017,-0.484044481741748,0.513167792394424],[0,0,0,0],[8.999999E+09,8.999999E+09,8.999999E+09,8.999999E+09,8.999999E+09,8.999999E+09]];
    LOCAL CONST Robtarget Tr_meulage_bavure_163 := [[121.2148671875,108.2778984375,76.8941953125],[0.536511367729273,-0.508895308767172,-0.463278982872616,0.488419595266758],[0,0,0,0],[8.999999E+09,8.999999E+09,8.999999E+09,8.999999E+09,8.999999E+09,8.999999E+09]];
    LOCAL CONST Robtarget Tr_meulage_bavure_164 := [[121.0355859375,105.851875,77.2852734375],[0.551014075847889,-0.525248015245261,-0.447423640567228,0.469372023623031],[0,0,0,0],[8.999999E+09,8.999999E+09,8.999999E+09,8.999999E+09,8.999999E+09,8.999999E+09]];
    LOCAL CONST Robtarget Tr_meulage_bavure_165 := [[120.6501015625,104.2673125,77.550546875],[0.561215077925295,-0.537255543772003,-0.435379296964472,0.454795541722075],[0,0,0,0],[8.999999E+09,8.999999E+09,8.999999E+09,8.999999E+09,8.999999E+09,8.999999E+09]];
    LOCAL CONST Robtarget Tr_meulage_bavure_166 := [[119.2860859375,99.6642578125,78.3301015625],[0.568131657701513,-0.545795974172248,-0.426689026395052,0.444150479960047],[0,0,0,0],[8.999999E+09,8.999999E+09,8.999999E+09,8.999999E+09,8.999999E+09,8.999999E+09]];
    LOCAL CONST Robtarget Tr_meulage_bavure_167 := [[119.1745,99.3745625,78.380109375],[0.572246399095995,-0.551267312460341,-0.421234034922241,0.437264561515736],[0,0,0,0],[8.999999E+09,8.999999E+09,8.999999E+09,8.999999E+09,8.999999E+09,8.999999E+09]];
    LOCAL CONST Robtarget Tr_meulage_bavure_168 := [[118.8790234375,98.2844296875,78.56371875],[0.573987539082143,-0.554047297755747,-0.418760242581797,0.433831483482718],[0,0,0,0],[8.999999E+09,8.999999E+09,8.999999E+09,8.999999E+09,8.999999E+09,8.999999E+09]];
    LOCAL CONST Robtarget Tr_meulage_bavure_169 := [[118.157640625,95.416125,79.0447734375],[0.573983618143378,-0.55473022025201,-0.418594701636289,0.433123151775819],[0,0,0,0],[8.999999E+09,8.999999E+09,8.999999E+09,8.999999E+09,8.999999E+09,8.999999E+09]];
    LOCAL CONST Robtarget Tr_meulage_bavure_170 := [[116.2935703125,88.042703125,80.2817421875],[0.57297772614128,-0.554056481807033,-0.419806644142427,0.434143204308734],[0,0,0,0],[8.999999E+09,8.999999E+09,8.999999E+09,8.999999E+09,8.999999E+09,8.999999E+09]];
    LOCAL CONST Robtarget Tr_meulage_bavure_171 := [[114.755921875,82.019671875,81.29271875],[0.571717009968474,-0.552766647784409,-0.421427712389544,0.435875414355996],[0,0,0,0],[8.999999E+09,8.999999E+09,8.999999E+09,8.999999E+09,8.999999E+09,8.999999E+09]];
    LOCAL CONST Robtarget Tr_meulage_bavure_172 := [[113.9568515625,79.0110859375,81.7988515625],[0.570741800658552,-0.551441542644947,-0.422751067890472,0.437547205023482],[0,0,0,0],[8.999999E+09,8.999999E+09,8.999999E+09,8.999999E+09,8.999999E+09,8.999999E+09]];
    LOCAL CONST Robtarget Tr_meulage_bavure_173 := [[113.0946953125,75.3961171875,82.40340625],[0.570291513227631,-0.550365440948714,-0.42346522249667,0.438796851271419],[0,0,0,0],[8.999999E+09,8.999999E+09,8.999999E+09,8.999999E+09,8.999999E+09,8.999999E+09]];
    LOCAL CONST Robtarget Tr_meulage_bavure_174 := [[111.866328125,70.247671875,83.2644296875],[0.570348548058846,-0.549558809715741,-0.423589079077199,0.439613398883058],[0,0,0,0],[8.999999E+09,8.999999E+09,8.999999E+09,8.999999E+09,8.999999E+09,8.999999E+09]];
    LOCAL CONST Robtarget Tr_meulage_bavure_175 := [[110.6963359375,65.5621796875,84.0499453125],[0.570730246257275,-0.548911775606505,-0.423339407549893,0.440166553276063],[0,0,0,0],[8.999999E+09,8.999999E+09,8.999999E+09,8.999999E+09,8.999999E+09,8.999999E+09]];
    LOCAL CONST Robtarget Tr_meulage_bavure_176 := [[109.079578125,59.30018359375,85.1016953125],[0.571202054662466,-0.548242644424327,-0.422999981438244,0.440714455500661],[0,0,0,0],[8.999999E+09,8.999999E+09,8.999999E+09,8.999999E+09,8.999999E+09,8.999999E+09]];
    LOCAL CONST Robtarget Tr_meulage_bavure_177 := [[108.9664609375,58.84338671875,85.1782421875],[0.571586602148422,-0.547413255173719,-0.422783831775528,0.441453639574685],[0,0,0,0],[8.999999E+09,8.999999E+09,8.999999E+09,8.999999E+09,8.999999E+09,8.999999E+09]];
    LOCAL CONST Robtarget Tr_meulage_bavure_178 := [[108.955265625,58.79690625,85.186015625],[0.571783729021885,-0.546395389519627,-0.422798655774579,0.44244405546095],[0,0,0,0],[8.999999E+09,8.999999E+09,8.999999E+09,8.999999E+09,8.999999E+09,8.999999E+09]];
    LOCAL CONST Robtarget Tr_meulage_bavure_179 := [[108.8861484375,58.48816015625,85.237484375],[0.571804532785428,-0.545228995882672,-0.423022019077319,0.443640946837146],[0,0,0,0],[8.999999E+09,8.999999E+09,8.999999E+09,8.999999E+09,8.999999E+09,8.999999E+09]];
    LOCAL CONST Robtarget Tr_meulage_bavure_180 := [[108.3659921875,56.17127734375,85.623765625],[0.571743622766661,-0.544026549746596,-0.423331111733246,0.444898991721899],[0,0,0,0],[8.999999E+09,8.999999E+09,8.999999E+09,8.999999E+09,8.999999E+09,8.999999E+09]];
    LOCAL CONST Robtarget Tr_meulage_bavure_181 := [[107.2515,51.11757421875,86.46559375],[0.571723754577021,-0.542919591600209,-0.423572858317666,0.446045176193644],[0,0,0,0],[8.999999E+09,8.999999E+09,8.999999E+09,8.999999E+09,8.999999E+09,8.999999E+09]];
    LOCAL CONST Robtarget Tr_meulage_bavure_182 := [[106.8913046875,49.38673828125,86.753125],[0.57185084902882,-0.542004843250663,-0.423621006211622,0.446948094809783],[0,0,0,0],[8.999999E+09,8.999999E+09,8.999999E+09,8.999999E+09,8.999999E+09,8.999999E+09]];
    LOCAL CONST Robtarget Tr_meulage_bavure_183 := [[105.4295703125,42.1545625,87.9529609375],[0.572163879538567,-0.54133606056187,-0.423427631567382,0.447540842060218],[0,0,0,0],[8.999999E+09,8.999999E+09,8.999999E+09,8.999999E+09,8.999999E+09,8.999999E+09]];
    LOCAL CONST Robtarget Tr_meulage_bavure_184 := [[104.96234375,39.9378984375,88.3214140625],[0.572662934443544,-0.540892920348453,-0.422998598388813,0.447843943793517],[0,0,0,0],[8.999999E+09,8.999999E+09,8.999999E+09,8.999999E+09,8.999999E+09,8.999999E+09]];
    LOCAL CONST Robtarget Tr_meulage_bavure_185 := [[103.34834375,32.7544296875,89.519109375],[0.573316399050442,-0.540619687732112,-0.422378039357179,0.447923488650745],[0,0,0,0],[8.999999E+09,8.999999E+09,8.999999E+09,8.999999E+09,8.999999E+09,8.999999E+09]];
    LOCAL CONST Robtarget Tr_meulage_bavure_186 := [[102.9133203125,30.917435546875,89.8262109375],[0.574079974065266,-0.540464438411367,-0.421621650539237,0.447845462170243],[0,0,0,0],[8.999999E+09,8.999999E+09,8.999999E+09,8.999999E+09,8.999999E+09,8.999999E+09]];
    LOCAL CONST Robtarget Tr_meulage_bavure_187 := [[102.3198671875,28.950740234375,90.159671875],[0.574938453136106,-0.540360123954557,-0.420757717877379,0.447682537510563],[0,0,0,0],[8.999999E+09,8.999999E+09,8.999999E+09,8.999999E+09,8.999999E+09,8.999999E+09]];
    LOCAL CONST Robtarget Tr_meulage_bavure_188 := [[100.5611171875,21.49590625,91.4056875],[0.57586541362976,-0.540262447091545,-0.41982170950574,0.447487704719759],[0,0,0,0],[8.999999E+09,8.999999E+09,8.999999E+09,8.999999E+09,8.999999E+09,8.999999E+09]];
    LOCAL CONST Robtarget Tr_meulage_bavure_189 := [[99.1413046875,15.9081181640625,92.343359375],[0.576836857947901,-0.54010804335628,-0.418850256949418,0.447333212569837],[0,0,0,0],[8.999999E+09,8.999999E+09,8.999999E+09,8.999999E+09,8.999999E+09,8.999999E+09]];
    LOCAL CONST Robtarget Tr_meulage_bavure_190 := [[97.671234375,9.9731259765625,93.33790625],[0.577818555474841,-0.539821853180802,-0.417892766417148,0.447307187013171],[0,0,0,0],[8.999999E+09,8.999999E+09,8.999999E+09,8.999999E+09,8.999999E+09,8.999999E+09]];
    LOCAL CONST Robtarget Tr_meulage_bavure_191 := [[96.315671875,4.5503349609375,94.247078125],[0.57876633120142,-0.539335240943723,-0.417007429523301,0.44749506753281],[0,0,0,0],[8.999999E+09,8.999999E+09,8.999999E+09,8.999999E+09,8.999999E+09,8.999999E+09]];
    LOCAL CONST Robtarget Tr_meulage_bavure_192 := [[95.476421875,1.26134619140625,94.799125],[0.57965737820399,-0.538578459667489,-0.416229841284663,0.447976880988311],[0,0,0,0],[8.999999E+09,8.999999E+09,8.999999E+09,8.999999E+09,8.999999E+09,8.999999E+09]];
    LOCAL CONST Robtarget Tr_meulage_bavure_193 := [[94.2034375,-3.87585083007813,95.6600078125],[0.580468138623368,-0.537535447518981,-0.415585102220813,0.448777679386808],[0,0,0,0],[8.999999E+09,8.999999E+09,8.999999E+09,8.999999E+09,8.999999E+09,8.999999E+09]];
    LOCAL CONST Robtarget Tr_meulage_bavure_194 := [[93.4653828125,-6.86782177734375,96.161265625],[0.581211148700069,-0.536201724430509,-0.415057740846841,0.449898191936366],[0,0,0,0],[8.999999E+09,8.999999E+09,8.999999E+09,8.999999E+09,8.999999E+09,8.999999E+09]];
    LOCAL CONST Robtarget Tr_meulage_bavure_195 := [[93.03571875,-8.293291015625,96.4029453125],[0.581921235213521,-0.534601662473156,-0.414603251728508,0.451301320787625],[0,0,0,0],[8.999999E+09,8.999999E+09,8.999999E+09,8.999999E+09,8.999999E+09,8.999999E+09]];
    LOCAL CONST Robtarget Tr_meulage_bavure_196 := [[92.75209375,-9.66555859375,96.6308359375],[0.582627239178533,-0.532812561607145,-0.414174409946529,0.452897154447097],[0,0,0,0],[8.999999E+09,8.999999E+09,8.999999E+09,8.999999E+09,8.999999E+09,8.999999E+09]];
    LOCAL CONST Robtarget Tr_meulage_bavure_197 := [[91.868546875,-13.3815673828125,97.2521875],[0.583400929149593,-0.530909318316545,-0.413681976941128,0.454583186607395],[0,0,0,0],[8.999999E+09,8.999999E+09,8.999999E+09,8.999999E+09,8.999999E+09,8.999999E+09]];
    LOCAL CONST Robtarget Tr_meulage_bavure_198 := [[91.1975390625,-16.1767421875,97.7198046875],[0.584323972321873,-0.529036620304723,-0.413018551523047,0.456181351925249],[0,0,0,0],[8.999999E+09,8.999999E+09,8.999999E+09,8.999999E+09,8.999999E+09,8.999999E+09]];
    LOCAL CONST Robtarget Tr_meulage_bavure_199 := [[90.400828125,-19.07030078125,98.2076171875],[0.585504545277529,-0.527368724720213,-0.412049765545176,0.457473109986255],[0,0,0,0],[8.999999E+09,8.999999E+09,8.999999E+09,8.999999E+09,8.999999E+09,8.999999E+09]];
    LOCAL CONST Robtarget Tr_meulage_bavure_200 := [[90.1165078125,-20.48877734375,98.442859375],[0.58710208608771,-0.526094256027421,-0.410590732569948,0.458204348096007],[0,0,0,0],[8.999999E+09,8.999999E+09,8.999999E+09,8.999999E+09,8.999999E+09,8.999999E+09]];
    LOCAL CONST Robtarget Tr_meulage_bavure_201 := [[88.447046875,-27.55845703125,99.6245546875],[0.589267826176401,-0.525459715350137,-0.408458118350407,0.458058382884908],[0,0,0,0],[8.999999E+09,8.999999E+09,8.999999E+09,8.999999E+09,8.999999E+09,8.999999E+09]];
    LOCAL CONST Robtarget Tr_meulage_bavure_202 := [[87.9321953125,-29.5916171875,99.965671875],[0.592145232368807,-0.525657015729735,-0.40547898504019,0.456766371669125],[0,0,0,0],[8.999999E+09,8.999999E+09,8.999999E+09,8.999999E+09,8.999999E+09,8.999999E+09]];
    LOCAL CONST Robtarget Tr_meulage_bavure_203 := [[87.0540234375,-33.175,100.5658125],[0.595778454978412,-0.526807509657832,-0.401578824579948,0.454154519960593],[0,0,0,0],[8.999999E+09,8.999999E+09,8.999999E+09,8.999999E+09,8.999999E+09,8.999999E+09]];
    LOCAL CONST Robtarget Tr_meulage_bavure_204 := [[86.617703125,-34.7503046875,100.8314765625],[0.600011317781909,-0.528857089473312,-0.396898155474074,0.450298180796583],[0,0,0,0],[8.999999E+09,8.999999E+09,8.999999E+09,8.999999E+09,8.999999E+09,8.999999E+09]];
    LOCAL CONST Robtarget Tr_meulage_bavure_205 := [[86.5871171875,-35.3041328125,100.920375],[0.604403471908682,-0.531494710693008,-0.391906523740372,0.445667019533444],[0,0,0,0],[8.999999E+09,8.999999E+09,8.999999E+09,8.999999E+09,8.999999E+09,8.999999E+09]];
    LOCAL CONST Robtarget Tr_meulage_bavure_206 := [[84.5125859375,-43.52753515625,102.29978125],[0.608231391444022,-0.534160768003874,-0.387434557286997,0.441159055452122],[0,0,0,0],[8.999999E+09,8.999999E+09,8.999999E+09,8.999999E+09,8.999999E+09,8.999999E+09]];
    LOCAL CONST Robtarget Tr_meulage_bavure_207 := [[84.31575,-44.277890625,102.425921875],[0.610673083228898,-0.536183109466185,-0.384485475865825,0.437900647854185],[0,0,0,0],[8.999999E+09,8.999999E+09,8.999999E+09,8.999999E+09,8.999999E+09,8.999999E+09]];
    LOCAL CONST Robtarget Tr_meulage_bavure_208 := [[84.095765625,-45.01173828125,102.550296875],[0.611144670130719,-0.53708119050953,-0.383807914053311,0.43673501357428],[0,0,0,0],[8.999999E+09,8.999999E+09,8.999999E+09,8.999999E+09,8.999999E+09,8.999999E+09]];
    LOCAL CONST Robtarget Tr_meulage_bavure_209 := [[83.927359375,-45.7833984375,102.6787734375],[0.609582149012711,-0.536800821583791,-0.385502212118417,0.437769946437418],[0,0,0,0],[8.999999E+09,8.999999E+09,8.999999E+09,8.999999E+09,8.999999E+09,8.999999E+09]];
    LOCAL CONST Robtarget Tr_meulage_bavure_210 := [[82.6511796875,-50.629109375,103.4935703125],[0.606453233802241,-0.535717385476319,-0.388988996664023,0.440350903920429],[0,0,0,0],[8.999999E+09,8.999999E+09,8.999999E+09,8.999999E+09,8.999999E+09,8.999999E+09]];
    LOCAL CONST Robtarget Tr_meulage_bavure_211 := [[82.519625,-51.10901171875,103.574453125],[0.602490208344315,-0.534425214560469,-0.393364180284696,0.443463482780904],[0,0,0,0],[8.999999E+09,8.999999E+09,8.999999E+09,8.999999E+09,8.999999E+09,8.999999E+09]];
    LOCAL CONST Robtarget Tr_meulage_bavure_212 := [[82.23215625,-52.15374609375,103.750578125],[0.598353690470349,-0.533438476326052,-0.397838325404641,0.446252081132049],[0,0,0,0],[8.999999E+09,8.999999E+09,8.999999E+09,8.999999E+09,8.999999E+09,8.999999E+09]];
    LOCAL CONST Robtarget Tr_meulage_bavure_213 := [[80.96809375,-56.879765625,104.5459609375],[0.594453264770159,-0.533039687908605,-0.401946106019189,0.448255881137556],[0,0,0,0],[8.999999E+09,8.999999E+09,8.999999E+09,8.999999E+09,8.999999E+09,8.999999E+09]];
    LOCAL CONST Robtarget Tr_meulage_bavure_214 := [[80.826515625,-57.4200546875,104.63678125],[0.590936299733153,-0.533276055492859,-0.405538848299835,0.449387561927685],[0,0,0,0],[8.999999E+09,8.999999E+09,8.999999E+09,8.999999E+09,8.999999E+09,8.999999E+09]];
    LOCAL CONST Robtarget Tr_meulage_bavure_215 := [[80.538625,-58.65389453125,104.842890625],[0.587775956073556,-0.534038288923852,-0.408668947838413,0.449791309940228],[0,0,0,0],[8.999999E+09,8.999999E+09,8.999999E+09,8.999999E+09,8.999999E+09,8.999999E+09]];
    LOCAL CONST Robtarget Tr_meulage_bavure_216 := [[77.7072890625,-69.790859375,106.7118203125],[0.584880047504568,-0.535178775747625,-0.411457257671205,0.449668692628271],[0,0,0,0],[8.999999E+09,8.999999E+09,8.999999E+09,8.999999E+09,8.999999E+09,8.999999E+09]];
    LOCAL CONST Robtarget Tr_meulage_bavure_217 := [[77.4994375,-70.47690625,106.828171875],[0.582186390544942,-0.536527501727881,-0.413995629070758,0.44922696453374],[0,0,0,0],[8.999999E+09,8.999999E+09,8.999999E+09,8.999999E+09,8.999999E+09,8.999999E+09]];
    LOCAL CONST Robtarget Tr_meulage_bavure_218 := [[77.3509765625,-71.191265625,106.9468359375],[0.579655984902404,-0.53798853557682,-0.416339518721138,0.448585198045793],[0,0,0,0],[8.999999E+09,8.999999E+09,8.999999E+09,8.999999E+09,8.999999E+09,8.999999E+09]];
    LOCAL CONST Robtarget Tr_meulage_bavure_219 := [[73.7572421875,-85.6021640625,109.362609375],[0.577297428997296,-0.539499037529054,-0.418490313719828,0.447810589759796],[0,0,0,0],[8.999999E+09,8.999999E+09,8.999999E+09,8.999999E+09,8.999999E+09,8.999999E+09]];
    LOCAL CONST Robtarget Tr_meulage_bavure_220 := [[73.654265625,-86.003609375,109.4300078125],[0.575135058868535,-0.541011921967839,-0.420431192102304,0.446948964711171],[0,0,0,0],[8.999999E+09,8.999999E+09,8.999999E+09,8.999999E+09,8.999999E+09,8.999999E+09]];
    LOCAL CONST Robtarget Tr_meulage_bavure_221 := [[73.5890078125,-86.1839140625,109.4609765625],[0.573176314138948,-0.542519003484333,-0.422155957326694,0.446011649468978],[0,0,0,0],[8.999999E+09,8.999999E+09,8.999999E+09,8.999999E+09,8.999999E+09,8.999999E+09]];
    LOCAL CONST Robtarget Tr_meulage_bavure_222 := [[73.5377265625,-86.400109375,109.497125],[0.571435605210462,-0.543986257566255,-0.423656591554264,0.445034148250937],[0,0,0,0],[8.999999E+09,8.999999E+09,8.999999E+09,8.999999E+09,8.999999E+09,8.999999E+09]];
    LOCAL CONST Robtarget Tr_meulage_bavure_223 := [[73.4722890625,-86.6506171875,109.5392265625],[0.569894534732582,-0.545393930897377,-0.424956591008785,0.444046816428666],[0,0,0,0],[8.999999E+09,8.999999E+09,8.999999E+09,8.999999E+09,8.999999E+09,8.999999E+09]];
    LOCAL CONST Robtarget Tr_meulage_bavure_224 := [[73.437984375,-86.74984375,109.5562109375],[0.56851740875469,-0.546728323914363,-0.426096374532899,0.443077843479635],[0,0,0,0],[8.999999E+09,8.999999E+09,8.999999E+09,8.999999E+09,8.999999E+09,8.999999E+09]];
    LOCAL CONST Robtarget Tr_meulage_bavure_225 := [[71.680578125,-94.1251015625,110.7895625],[0.567277659922664,-0.547959568713347,-0.427110699996483,0.442168313605423],[0,0,0,0],[8.999999E+09,8.999999E+09,8.999999E+09,8.999999E+09,8.999999E+09,8.999999E+09]];
    LOCAL CONST Robtarget Tr_meulage_bavure_226 := [[70.7323671875,-98.0152734375,111.440890625],[0.566125626783543,-0.549083820697172,-0.428052876338697,0.441338268911392],[0,0,0,0],[8.999999E+09,8.999999E+09,8.999999E+09,8.999999E+09,8.999999E+09,8.999999E+09]];
    LOCAL CONST Robtarget Tr_meulage_bavure_227 := [[70.6430390625,-98.3930703125,111.5040390625],[0.565026931471466,-0.550095219835362,-0.428960891945603,0.440604549462959],[0,0,0,0],[8.999999E+09,8.999999E+09,8.999999E+09,8.999999E+09,8.999999E+09,8.999999E+09]];
    LOCAL CONST Robtarget Tr_meulage_bavure_228 := [[67.9664765625,-109.1046171875,113.2998671875],[0.563943167242867,-0.551005348350713,-0.42987289697444,0.439966479013794],[0,0,0,0],[8.999999E+09,8.999999E+09,8.999999E+09,8.999999E+09,8.999999E+09,8.999999E+09]];
    LOCAL CONST Robtarget Tr_meulage_bavure_229 := [[67.89590625,-109.4032578125,113.3497890625],[0.562839647758574,-0.551826224711239,-0.430822831213495,0.43942125203173],[0,0,0,0],[8.999999E+09,8.999999E+09,8.999999E+09,8.999999E+09,8.999999E+09,8.999999E+09]];
    LOCAL CONST Robtarget Tr_meulage_bavure_230 := [[64.87401953125,-121.8640078125,115.4355078125],[0.561701852391063,-0.552574260009182,-0.431822576003232,0.438955554754334],[0,0,0,0],[8.999999E+09,8.999999E+09,8.999999E+09,8.999999E+09,8.999999E+09,8.999999E+09]];
    LOCAL CONST Robtarget Tr_meulage_bavure_231 := [[63.45353515625,-127.771390625,116.4238671875],[0.560508148890272,-0.553290208333834,-0.432885370705927,0.438532571445149],[0,0,0,0],[8.999999E+09,8.999999E+09,8.999999E+09,8.999999E+09,8.999999E+09,8.999999E+09]];
    LOCAL CONST Robtarget Tr_meulage_bavure_232 := [[63.3378203125,-128.2375625,116.5019921875],[0.559273417750795,-0.554022254393372,-0.433984646298402,0.438098062779878],[0,0,0,0],[8.999999E+09,8.999999E+09,8.999999E+09,8.999999E+09,8.999999E+09,8.999999E+09]];
    LOCAL CONST Robtarget Tr_meulage_bavure_233 := [[62.84611328125,-130.287046875,116.84484375],[0.558091793023811,-0.554907957852992,-0.434990336014533,0.437486132860063],[0,0,0,0],[8.999999E+09,8.999999E+09,8.999999E+09,8.999999E+09,8.999999E+09,8.999999E+09]];
    LOCAL CONST Robtarget Tr_meulage_bavure_234 := [[61.62488671875,-135.58378125,117.729109375],[0.557177855275096,-0.556207808319746,-0.435616363233738,0.436376094256091],[0,0,0,0],[8.999999E+09,8.999999E+09,8.999999E+09,8.999999E+09,8.999999E+09,8.999999E+09]];
    LOCAL CONST Robtarget Tr_meulage_bavure_235 := [[60.569234375,-140.050203125,118.4757109375],[0.556944476421682,-0.558345521652502,-0.435323434413339,0.434231086041235],[0,0,0,0],[8.999999E+09,8.999999E+09,8.999999E+09,8.999999E+09,8.999999E+09,8.999999E+09]];
    LOCAL CONST Robtarget Tr_meulage_bavure_236 := [[60.43681640625,-140.897046875,118.61478125],[0.557975694412541,-0.561963629776834,-0.433310146594765,0.430235191623037],[0,0,0,0],[8.999999E+09,8.999999E+09,8.999999E+09,8.999999E+09,8.999999E+09,8.999999E+09]];
    LOCAL CONST Robtarget Tr_meulage_bavure_237 := [[58.879875,-147.847921875,119.7735234375],[0.561032915136402,-0.567863867276577,-0.428464006266995,0.423309923943296],[0,0,0,0],[8.999999E+09,8.999999E+09,8.999999E+09,8.999999E+09,8.999999E+09,8.999999E+09]];
    LOCAL CONST Robtarget Tr_meulage_bavure_238 := [[58.4683203125,-149.7818125,120.0951171875],[0.56686707752109,-0.576856078116111,-0.419487969328714,0.412223998757557],[0,0,0,0],[8.999999E+09,8.999999E+09,8.999999E+09,8.999999E+09,8.999999E+09,8.999999E+09]];
    LOCAL CONST Robtarget Tr_meulage_bavure_239 := [[58.34700390625,-150.2285,120.170359375],[0.576094073640307,-0.589632704144517,-0.404901969259845,0.395604964338468],[0,0,0,0],[8.999999E+09,8.999999E+09,8.999999E+09,8.999999E+09,8.999999E+09,8.999999E+09]];
    LOCAL CONST Robtarget Tr_meulage_bavure_240 := [[58.01381640625,-150.72125,120.260671875],[0.589149999527341,-0.606676748512503,-0.38287957710617,0.371818275917459],[0,0,0,0],[8.999999E+09,8.999999E+09,8.999999E+09,8.999999E+09,8.999999E+09,8.999999E+09]];
    LOCAL CONST Robtarget Tr_meulage_bavure_241 := [[56.1310703125,-154.04634375,120.8567109375],[0.60610616428059,-0.628140585106259,-0.351121406680601,0.338804487476292],[0,0,0,0],[8.999999E+09,8.999999E+09,8.999999E+09,8.999999E+09,8.999999E+09,8.999999E+09]];
    LOCAL CONST Robtarget Tr_meulage_bavure_242 := [[54.48117578125,-154.702421875,121.0211875],[0.626326189084628,-0.653442669948181,-0.306906737478566,0.294170760695181],[0,0,0,0],[8.999999E+09,8.999999E+09,8.999999E+09,8.999999E+09,8.999999E+09,8.999999E+09]];
    LOCAL CONST Robtarget Tr_meulage_bavure_243 := [[53.3359765625,-155.232765625,121.147234375],[0.647671429312515,-0.680363137621262,-0.248410350767661,0.236474138649287],[0,0,0,0],[8.999999E+09,8.999999E+09,8.999999E+09,8.999999E+09,8.999999E+09,8.999999E+09]];
    LOCAL CONST Robtarget Tr_meulage_bavure_244 := [[52.95303125,-155.318125,121.1748046875],[0.66606212123288,-0.704598438139302,-0.177859430635197,0.16813183685589],[0,0,0,0],[8.999999E+09,8.999999E+09,8.999999E+09,8.999999E+09,8.999999E+09,8.999999E+09]];
    LOCAL CONST Robtarget Tr_meulage_bavure_245 := [[51.18946875,-155.148484375,121.2125859375],[0.677377245040288,-0.721648574729892,-0.104096476827729,0.0977104191168941],[0,0,0,0],[8.999999E+09,8.999999E+09,8.999999E+09,8.999999E+09,8.999999E+09,8.999999E+09]];
    LOCAL CONST Robtarget Tr_meulage_bavure_246 := [[49.75246875,-154.979265625,121.2384609375],[0.680867811392423,-0.730482503056316,-0.0388069747920954,0.0361711880611846],[0,0,0,0],[8.999999E+09,8.999999E+09,8.999999E+09,8.999999E+09,8.999999E+09,8.999999E+09]];
    LOCAL CONST Robtarget Tr_meulage_bavure_247 := [[46.9879375,-154.264109375,121.226484375],[0.679212480214634,-0.733790855497135,0.0109193437756427,-0.010107177695947],[0,0,0,0],[8.999999E+09,8.999999E+09,8.999999E+09,8.999999E+09,8.999999E+09,8.999999E+09]];
    LOCAL CONST Robtarget Tr_meulage_bavure_248 := [[43.8973359375,-153.507984375,121.2199765625],[0.675553665647016,-0.734818107605313,0.0445950998202359,-0.0409984223873215],[0,0,0,0],[8.999999E+09,8.999999E+09,8.999999E+09,8.999999E+09,8.999999E+09,8.999999E+09]];
    LOCAL CONST Robtarget Tr_meulage_bavure_249 := [[42.30314453125,-153.179359375,121.22634375],[0.671734986232103,-0.735493769781421,0.0653003886716209,-0.0596396019755793],[0,0,0,0],[8.999999E+09,8.999999E+09,8.999999E+09,8.999999E+09,8.999999E+09,8.999999E+09]];
    LOCAL CONST Robtarget Tr_meulage_bavure_250 := [[33.237171875,-151.070265625,121.2245078125],[0.668410818492601,-0.736494966158005,0.0769632061451827,-0.0698484605830694],[0,0,0,0],[8.999999E+09,8.999999E+09,8.999999E+09,8.999999E+09,8.999999E+09,8.999999E+09]];
    LOCAL CONST Robtarget Tr_meulage_bavure_251 := [[31.8516875,-150.748828125,121.2243671875],[0.66563456824769,-0.737855576781333,0.0830144626649375,-0.0748890402852717],[0,0,0,0],[8.999999E+09,8.999999E+09,8.999999E+09,8.999999E+09,8.999999E+09,8.999999E+09]];
    LOCAL CONST Robtarget Tr_meulage_bavure_252 := [[31.44025,-150.64884375,121.223609375],[0.663269281737297,-0.739407547192561,0.0860099195518451,-0.0771533071038268],[0,0,0,0],[8.999999E+09,8.999999E+09,8.999999E+09,8.999999E+09,8.999999E+09,8.999999E+09]];
    LOCAL CONST Robtarget Tr_meulage_bavure_253 := [[31.111515625,-150.569265625,121.223046875],[0.661188430877681,-0.740984999149361,0.0875597893900946,-0.078130488230231],[0,0,0,0],[8.999999E+09,8.999999E+09,8.999999E+09,8.999999E+09,8.999999E+09,8.999999E+09]];
    LOCAL CONST Robtarget Tr_meulage_bavure_254 := [[26.904798828125,-149.5583125,121.217078125],[0.659312478248861,-0.74248886009966,0.0885295472553769,-0.0786121359334034],[0,0,0,0],[8.999999E+09,8.999999E+09,8.999999E+09,8.999999E+09,8.999999E+09,8.999999E+09]];
    LOCAL CONST Robtarget Tr_meulage_bavure_255 := [[18.802130859375,-147.605609375,121.204703125],[0.657605383733481,-0.743860250521355,0.0893636512700392,-0.0790014228399371],[0,0,0,0],[8.999999E+09,8.999999E+09,8.999999E+09,8.999999E+09,8.999999E+09,8.999999E+09]];
    LOCAL CONST Robtarget Tr_meulage_bavure_256 := [[18.244751953125,-147.461125,121.2022421875],[0.656059252329324,-0.74508184642979,0.0901852173954756,-0.07940986158654],[0,0,0,0],[8.999999E+09,8.999999E+09,8.999999E+09,8.999999E+09,8.999999E+09,8.999999E+09]];
    LOCAL CONST Robtarget Tr_meulage_bavure_257 := [[16.867578125,-147.132546875,121.2006640625],[0.654673036163601,-0.746144174916212,0.0910496521630891,-0.0798877136981507],[0,0,0,0],[8.999999E+09,8.999999E+09,8.999999E+09,8.999999E+09,8.999999E+09,8.999999E+09]];
    LOCAL CONST Robtarget Tr_meulage_bavure_258 := [[13.8791943359375,-146.41165625,121.195984375],[0.653452722206137,-0.747037566231934,0.0919822372351747,-0.0804591978139884],[0,0,0,0],[8.999999E+09,8.999999E+09,8.999999E+09,8.999999E+09,8.999999E+09,8.999999E+09]];
    LOCAL CONST Robtarget Tr_meulage_bavure_259 := [[8.6903837890625,-145.144078125,121.1853515625],[0.652401793980607,-0.747765759772904,0.0929561638956427,-0.081101290470281],[0,0,0,0],[8.999999E+09,8.999999E+09,8.999999E+09,8.999999E+09,8.999999E+09,8.999999E+09]];
    LOCAL CONST Robtarget Tr_meulage_bavure_260 := [[4.88120556640625,-144.255875,121.1842578125],[0.651528115643831,-0.748336616273692,0.0939082381760919,-0.0817598071934037],[0,0,0,0],[8.999999E+09,8.999999E+09,8.999999E+09,8.999999E+09,8.999999E+09,8.999999E+09]];
    LOCAL CONST Robtarget Tr_meulage_bavure_261 := [[-2.90349291992188,-142.3619375,121.1695390625],[0.650851982241957,-0.748757213899782,0.0947303753560355,-0.0823437176089133],[0,0,0,0],[8.999999E+09,8.999999E+09,8.999999E+09,8.999999E+09,8.999999E+09,8.999999E+09]];
    LOCAL CONST Robtarget Tr_meulage_bavure_262 := [[-3.63015795898438,-142.170828125,121.165890625],[0.650386942995498,-0.749046209994587,0.0952919899840636,-0.0827407778461901],[0,0,0,0],[8.999999E+09,8.999999E+09,8.999999E+09,8.999999E+09,8.999999E+09,8.999999E+09]];
    LOCAL CONST Robtarget Tr_meulage_bavure_263 := [[-4.46912939453125,-141.956,121.162609375],[0.650144078875515,-0.74921879246872,0.0954879630957082,-0.082860887146194],[0,0,0,0],[8.999999E+09,8.999999E+09,8.999999E+09,8.999999E+09,8.999999E+09,8.999999E+09]];
    LOCAL CONST Robtarget Tr_meulage_bavure_264 := [[-4.524146484375,-141.808765625,121.1412890625],[0.650124247046936,-0.749282815679199,0.0952829329367833,-0.0826733827811042],[0,0,0,0],[8.999999E+09,8.999999E+09,8.999999E+09,8.999999E+09,8.999999E+09,8.999999E+09]];
    LOCAL CONST Robtarget Tr_meulage_bavure_265 := [[-6.66910888671875,-141.397,121.1546796875],[0.650316062659858,-0.749235522785154,0.0947322421207195,-0.082225010466505],[0,0,0,0],[8.999999E+09,8.999999E+09,8.999999E+09,8.999999E+09,8.999999E+09,8.999999E+09]];
    LOCAL CONST Robtarget Tr_meulage_bavure_266 := [[-12.70651953125,-139.931890625,121.1438515625],[0.650698242406178,-0.749063372137148,0.0939761516043519,-0.0816354382708385],[0,0,0,0],[8.999999E+09,8.999999E+09,8.999999E+09,8.999999E+09,8.999999E+09,8.999999E+09]];
    LOCAL CONST Robtarget Tr_meulage_bavure_267 := [[-14.51728515625,-139.50603125,121.1427578125],[0.65124173587056,-0.748753806196818,0.093183497744998,-0.0810479790869888],[0,0,0,0],[8.999999E+09,8.999999E+09,8.999999E+09,8.999999E+09,8.999999E+09,8.999999E+09]];
    LOCAL CONST Robtarget Tr_meulage_bavure_268 := [[-14.9362265625,-139.405625,121.142203125],[0.651913321773216,-0.748303655818487,0.092501481106863,-0.0805861996643044],[0,0,0,0],[8.999999E+09,8.999999E+09,8.999999E+09,8.999999E+09,8.999999E+09,8.999999E+09]];
    LOCAL CONST Robtarget Tr_meulage_bavure_269 := [[-15.532115234375,-139.2733125,121.1430859375],[0.652687070827292,-0.747721091492607,0.0919986073345962,-0.0803057479915979],[0,0,0,0],[8.999999E+09,8.999999E+09,8.999999E+09,8.999999E+09,8.999999E+09,8.999999E+09]];
    LOCAL CONST Robtarget Tr_meulage_bavure_270 := [[-20.544951171875,-137.98059375,121.122015625],[0.653547423424678,-0.747027351415611,0.0916411576902467,-0.0801735604119725],[0,0,0,0],[8.999999E+09,8.999999E+09,8.999999E+09,8.999999E+09,8.999999E+09,8.999999E+09]];
    LOCAL CONST Robtarget Tr_meulage_bavure_271 := [[-28.533595703125,-136.09009375,121.1153203125],[0.654486498639298,-0.746255340131277,0.0913095230022755,-0.0800809679856642],[0,0,0,0],[8.999999E+09,8.999999E+09,8.999999E+09,8.999999E+09,8.999999E+09,8.999999E+09]];
    LOCAL CONST Robtarget Tr_meulage_bavure_272 := [[-29.160009765625,-135.94228125,121.114859375],[0.65549294105227,-0.745450396597255,0.0908410339861932,-0.079878764311678],[0,0,0,0],[8.999999E+09,8.999999E+09,8.999999E+09,8.999999E+09,8.999999E+09,8.999999E+09]];
    LOCAL CONST Robtarget Tr_meulage_bavure_273 := [[-29.947775390625,-135.74315625,121.1121875],[0.656552799646047,-0.744653727866067,0.090101557024869,-0.079441527388399],[0,0,0,0],[8.999999E+09,8.999999E+09,8.999999E+09,8.999999E+09,8.999999E+09,8.999999E+09]];
    LOCAL CONST Robtarget Tr_meulage_bavure_274 := [[-37.47444140625,-133.90090625,121.0961953125],[0.657643412862154,-0.743896375419463,0.0890368137734188,-0.0787132133118755],[0,0,0,0],[8.999999E+09,8.999999E+09,8.999999E+09,8.999999E+09,8.999999E+09,8.999999E+09]];
    LOCAL CONST Robtarget Tr_meulage_bavure_275 := [[-41.598703125,-132.783578125,121.07034375],[0.658732991419729,-0.743195631701016,0.0876916271219011,-0.0777256557930255],[0,0,0,0],[8.999999E+09,8.999999E+09,8.999999E+09,8.999999E+09,8.999999E+09,8.999999E+09]];
    LOCAL CONST Robtarget Tr_meulage_bavure_276 := [[-42.98394140625,-132.45828125,121.069578125],[0.659783704257721,-0.742558207918677,0.0861874669322046,-0.076579971222064],[0,0,0,0],[8.999999E+09,8.999999E+09,8.999999E+09,8.999999E+09,8.999999E+09,8.999999E+09]];
    LOCAL CONST Robtarget Tr_meulage_bavure_277 := [[-47.9850625,-131.286984375,121.0673203125],[0.660755664164215,-0.741987280938255,0.0846785262747031,-0.0754080525455051],[0,0,0,0],[8.999999E+09,8.999999E+09,8.999999E+09,8.999999E+09,8.999999E+09,8.999999E+09]];
    LOCAL CONST Robtarget Tr_meulage_bavure_278 := [[-50.09307421875,-130.8154453125,121.0698828125],[0.661616595398046,-0.741485689120522,0.0832966894234594,-0.0743243907102836],[0,0,0,0],[8.999999E+09,8.999999E+09,8.999999E+09,8.999999E+09,8.999999E+09,8.999999E+09]];
    LOCAL CONST Robtarget Tr_meulage_bavure_279 := [[-50.36609375,-130.7348125,121.0671171875],[0.662340618402317,-0.741058006277795,0.0821441199637836,-0.073418526962829],[0,0,0,0],[8.999999E+09,8.999999E+09,8.999999E+09,8.999999E+09,8.999999E+09,8.999999E+09]];
    LOCAL CONST Robtarget Tr_meulage_bavure_280 := [[-58.0085390625,-128.848421875,121.048375],[0.662908454855615,-0.740709166917427,0.0812949214712567,-0.0727560737561752],[0,0,0,0],[8.999999E+09,8.999999E+09,8.999999E+09,8.999999E+09,8.999999E+09,8.999999E+09]];
    LOCAL CONST Robtarget Tr_meulage_bavure_281 := [[-58.33327734375,-128.7690546875,121.047703125],[0.663320268102517,-0.740437081028021,0.0807690067497359,-0.0723568829605676],[0,0,0,0],[8.999999E+09,8.999999E+09,8.999999E+09,8.999999E+09,8.999999E+09,8.999999E+09]];
    LOCAL CONST Robtarget Tr_meulage_bavure_282 := [[-66.1873984375,-126.856109375,121.032515625],[0.663576594867529,-0.740253043442468,0.0805136842552313,-0.0721739639054629],[0,0,0,0],[8.999999E+09,8.999999E+09,8.999999E+09,8.999999E+09,8.999999E+09,8.999999E+09]];
    LOCAL CONST Robtarget Tr_meulage_bavure_283 := [[-67.37746875,-126.56565625,121.030125],[0.663701013889796,-0.740175399355127,0.0803302080706877,-0.072030549230553],[0,0,0,0],[8.999999E+09,8.999999E+09,8.999999E+09,8.999999E+09,8.999999E+09,8.999999E+09]];
    LOCAL CONST Robtarget Tr_meulage_bavure_284 := [[-68.239375,-126.3459921875,121.0269140625],[0.663740372974985,-0.740233915326161,0.0798503270541025,-0.0715988348598048],[0,0,0,0],[8.999999E+09,8.999999E+09,8.999999E+09,8.999999E+09,8.999999E+09,8.999999E+09]];
    LOCAL CONST Robtarget Tr_meulage_bavure_285 := [[-71.43075,-125.597859375,121.025359375],[0.663750783199385,-0.740462237355982,0.0786296643100021,-0.0704836771350133],[0,0,0,0],[8.999999E+09,8.999999E+09,8.999999E+09,8.999999E+09,8.999999E+09,8.999999E+09]];
    LOCAL CONST Robtarget Tr_meulage_bavure_286 := [[-73.1835078125,-125.130421875,121.015546875],[0.663773723337364,-0.740878798348823,0.0763304215634768,-0.0683865272403772],[0,0,0,0],[8.999999E+09,8.999999E+09,8.999999E+09,8.999999E+09,8.999999E+09,8.999999E+09]];
    LOCAL CONST Robtarget Tr_meulage_bavure_287 := [[-74.887875,-124.7250625,121.013796875],[0.66381871802067,-0.741451673347551,0.072975813981589,-0.0653349544213194],[0,0,0,0],[8.999999E+09,8.999999E+09,8.999999E+09,8.999999E+09,8.999999E+09,8.999999E+09]];
    LOCAL CONST Robtarget Tr_meulage_bavure_288 := [[-76.6340234375,-124.3405390625,121.0168828125],[0.663853533715442,-0.742095637659054,0.0690867610247557,-0.0618026681627116],[0,0,0,0],[8.999999E+09,8.999999E+09,8.999999E+09,8.999999E+09,8.999999E+09,8.999999E+09]];
    LOCAL CONST Robtarget Tr_meulage_bavure_289 := [[-79.59890625,-123.7010078125,121.0242421875],[0.663817545178961,-0.742700195390393,0.0656065530820179,-0.0586384402277776],[0,0,0,0],[8.999999E+09,8.999999E+09,8.999999E+09,8.999999E+09,8.999999E+09,8.999999E+09]];
    LOCAL CONST Robtarget Tr_meulage_bavure_290 := [[-82.3600546875,-122.9909765625,121.012953125],[0.663662713934865,-0.74316497542136,0.0635424723426249,-0.0567448292636874],[0,0,0,0],[8.999999E+09,8.999999E+09,8.999999E+09,8.999999E+09,8.999999E+09,8.999999E+09]];
    LOCAL CONST Robtarget Tr_meulage_bavure_291 := [[-83.878234375,-122.83784375,121.0443515625],[0.663377042091491,-0.743429728116851,0.0635011947185109,-0.0566633713025535],[0,0,0,0],[8.999999E+09,8.999999E+09,8.999999E+09,8.999999E+09,8.999999E+09,8.999999E+09]];
    LOCAL CONST Robtarget Tr_meulage_bavure_292 := [[-85.91796875,-122.438421875,121.05584375],[0.662986108880681,-0.743495470208808,0.0653392274127663,-0.0582639731853293],[0,0,0,0],[8.999999E+09,8.999999E+09,8.999999E+09,8.999999E+09,8.999999E+09,8.999999E+09]];
    LOCAL CONST Robtarget Tr_meulage_bavure_293 := [[-88.750171875,-121.7826953125,121.055765625],[0.662574623350153,-0.743413895968023,0.0681375659302057,-0.0607282461722294],[0,0,0,0],[8.999999E+09,8.999999E+09,8.999999E+09,8.999999E+09,8.999999E+09,8.999999E+09]];
    LOCAL CONST Robtarget Tr_meulage_bavure_294 := [[-93.7918515625,-120.5591953125,121.0467265625],[0.662255165903041,-0.743290019194477,0.0705877125454274,-0.0628921095067969],[0,0,0,0],[8.999999E+09,8.999999E+09,8.999999E+09,8.999999E+09,8.999999E+09,8.999999E+09]];
    LOCAL CONST Robtarget Tr_meulage_bavure_295 := [[-96.5772578125,-119.9039140625,121.0450078125],[0.662133890932801,-0.743233056978546,0.0715531148197318,-0.0637454724047857],[0,0,0,0],[8.999999E+09,8.999999E+09,8.999999E+09,8.999999E+09,8.999999E+09,8.999999E+09]];
    !
    !Declaration des points de tronconnage

    !
    !Cycle
    LOCAL PROC Cycle()
        !
        Prise;
        !
        Meulage;
        !
        !
        Depose;
        !
    ENDPROC

    !Trajectoire de prise de la pièce
    LOCAL PROC PRISE()

		!
        !Trigger localisation
        LocalisationPieceTable 704 \model:=1;
        !
        !Approche
		MoveJ Reltool(PicKPosition,0,0,-100),V1000,Z0,Tool_Prehenseur1 \Wobj:=Wobj_vision;
		MoveL Reltool(PicKPosition,0,0,-50),V500,Z0,Tool_Prehenseur1 \Wobj:=Wobj_vision;
		MoveL Reltool(PicKPosition,0,0,-10),V200,Z0,Tool_Prehenseur1 \Wobj:=Wobj_vision;
		MoveL PicKPosition,V100,Fine,Tool_Prehenseur1 \Wobj:=Wobj_vision;

        !Fermeture pince
		Gripper_Close;
        !
		MoveL Reltool(PicKPosition,0,0,-100),V500,Z0,Tool_Prehenseur1 \Wobj:=Wobj_vision;

        !Trigger relocalisation
		LocalisationPiecePrehenseur 704 \model:=1,Ref;
        !
        PEO;
        !
    ENDPROC

    !Trajectoire de tronconnage
    LOCAL PROC Tronconnage()
        !
        !StartMotor1();
        !
        ConfJ \Off;
        ConfL \Off;


    ENDPROC


    !Trajectoire de meulage
    LOCAL PROC Meulage()
        !
        !StartMotor2();
        !

        ConfJ \Off;
        ConfL \Off;


        !---------- Meulage zone : 1 ------------

        !Approche PLAN

        Go_to_Meulage_Plan;
		Tool := ToolOffset(Tool_M1_D500_S0 \Z);

